(* Logix 5000 project; controller Almacen_1 vendor 1 type 14 code 235 rev 36.11; software revision 36.00 *)

TASK MainTask (continuous, watchdog 500 ms) : MainProgram, _02_Conveyor_1
TASK SafetyTask (periodic, rate 20 ms, priority 10, watchdog 20 ms, safety) : SafetyProgram

MODULES
   Local : vendor 1 type 14 code 235 (5069 0, rev 36.11)
      Logix_Principal : vendor 1 type 12 code 200 (Ethernet 10.12.143.10, rev 10.7, Output RPI 10 ms)
           Point_IO_Conveyor_1:2:I.4   // Sensor Piston Horizontal Extendido
           Point_IO_Conveyor_1:2:I.5   // Sensor Piston Horizontal Retraido
           Point_IO_Conveyor_1:2:I.6   // Sensor Inductivo Presencia en Zona de Vision (Actual Marcadora Laser)
           Point_IO_Conveyor_1:2:I.0   // Sensor difuso presencia lado B Almacen 2-1 (Robot)
           Point_IO_Conveyor_1:2:I.1   // Sensor difuso presencia lado B Almacen 2-2 (Robot)
           Point_IO_Conveyor_1:2:I.2   // Sensor Difuso Lado A CNC 3-1 (Centro-Marcadora Laser)
           Point_IO_Conveyor_1:2:I.3   // Sensor Difuso Lado A CNC 3-2 (Centro-Marcadora Laser)
           Point_IO_Conveyor_1:2:I.7   // Spare
           Point_IO_Conveyor_1:4:I.0   // Cambio de Dirección Extendido Lado A
           Point_IO_Conveyor_1:4:I.1   // Cambio de Dirección Retraido Lado A
           Point_IO_Conveyor_1:4:I.2   // Sensor 2 Posición Tope Corredizo Lado Almacen Izq
           Point_IO_Conveyor_1:4:I.3   // Sensor Inductivo Posición Lado B CNC
           Point_IO_Conveyor_1:4:I.6   // Sensor Límite Lado CNC Der
           Point_IO_Conveyor_1:4:I.7   // Sensor Posición Tope Corredizo Lado Almacen Der
           Point_IO_Conveyor_1:4:I.4   // Spare
           Point_IO_Conveyor_1:4:I.5   // Spare
           Point_IO_Conveyor_1:7:O.2   // Tope Piston CNC (Freno 5)
           Point_IO_Conveyor_1:7:O.3   // Tope Pison Marcadora Laser (Freno 06)
           Point_IO_Conveyor_1:7:O.4   // Subir Limit Switch
           Point_IO_Conveyor_1:7:O.5   // Tope Piston Cámara Visión
           Point_IO_Conveyor_1:7:O.6   // Sensor Límite Lado CNC Izq
           Point_IO_Conveyor_1:7:O.7   // Piston Cambio de Dirección Almacén
           Point_IO_Conveyor_1:7:O.0   // Piston Horizontal Para Salida de Pieza
           Point_IO_Conveyor_1:7:O.1   // Tope Piston Salida de Producto (Freno 8)
           Point_IO_Almacen1:2:I.5   // Boton Azul
           Point_IO_Almacen1:2:I.7   // Botón verde
           Point_IO_Almacen1:2:I.0   // Botón Verde Reset Vvula General Almacén 1
           Point_IO_Almacen1:3:O.0   // actuador posicionador horizontal lado derecho
           Point_IO_Almacen1:3:O.1   // actuador posicionador horizontal lado izquierdo
           Point_IO_Almacen1:3:O.2   // Actuador sencillo clamp abajo
           Point_IO_Almacen1:3:O.3   // Actuador Clamp arriba
           Point_IO_Almacen1:3:O.4   // actuador de giro direccion conveyor
           Point_IO_Almacen1:3:O.5   // actuador de giro direccion almacen
           Point_IO_Almacen1:3:O.6   // Posicion dejar pieza
           Point_IO_Almacen1:3:O.7   // Posicion tomar pieza
           Point_IO_Almacen1:4:O.0   // lampara LED verde botonera 1
           Point_IO_Almacen1:4:O.1   // RELEVADOR 1
           Point_IO_Almacen1:4:O.2   // RELEVADOR 2
           Point_IO_Almacen1:4:O.3   // RELEVADOR 3
           Point_IO_Almacen1:4:O.4   // RELEVADOR 4
           Point_IO_Almacen1:4:O.5   // RELEVADOR 5
           Point_IO_Almacen1:4:O.6   // RELEVADOR 6
           Point_IO_Almacen1:4:O.7   // SPARE
           Point_IO_Almacen1:5:O.0   // Luz Verde Almacen 1
           Point_IO_Almacen1:5:O.1   // Luz Ambar Almacen 1
           Point_IO_Almacen1:5:O.2   // Luz Roja Almacén 1
           Point_IO_Conveyor_1:1:I.2   // Boton negro Puerta
           Point_IO_Conveyor_1:1:I.3   // Boton Rojo Puerta
           Point_IO_Conveyor_1:1:I.4   // Auxiliar Scanner de Seguridad (Sin Conexión)
           Point_IO_Conveyor_1:1:I.6   // Sensor difuso presencia lado A Almacen 1-1
           Point_IO_Conveyor_1:1:I.7   // Sensor difuso presencia lado A Almacen 1-2
           Point_IO_Conveyor_1:1:I.0   // Spare
           Point_IO_Conveyor_1:1:I.1   // Spare
           Point_IO_Conveyor_1:1:I.5   // Spare
           Point_IO_Conveyor_1:3:I.2   // Sensor Piston Tope CNC
           Point_IO_Conveyor_1:3:I.3   // Sensor Piston Tope Marcadora Laser
           Point_IO_Conveyor_1:3:I.4   // Límit Switch Arriba
           Point_IO_Conveyor_1:3:I.5   // Sensor Piston Tope Camara Vision
           Point_IO_Conveyor_1:3:I.6   // Cambio de Dirección Extendido Lado B
           Point_IO_Conveyor_1:3:I.7   // Cambio de Dirección Retraido Lado B
           Point_IO_Conveyor_1:3:I.1   // Sensor Tope Piston Horizontal (Salida de conveyor)
           Point_IO_Conveyor_1:3:I.0   // Spare
           Point_IO_Conveyor_1:5:I.0   // Sensor Limit Switch Tope
           Point_IO_Conveyor_1:5:I.1   // Sensor Posición Tope Corredizo Lado Almacen Izq
           Point_IO_Conveyor_1:5:I.2   // Spare
           Point_IO_Conveyor_1:5:I.3   // Spare
           Point_IO_Conveyor_1:5:I.4   // Spare
           Point_IO_Conveyor_1:5:I.5   // Spare
           Point_IO_Conveyor_1:5:I.6   // Spare
           Point_IO_Conveyor_1:5:I.7   // Spare
           Point_IO_Conveyor_1:6:I.0   // Spare
           Point_IO_Conveyor_1:6:I.1   // Spare
           Point_IO_Conveyor_1:6:I.2   // Spare
           Point_IO_Conveyor_1:6:I.3   // Spare
           Point_IO_Conveyor_1:6:I.4   // Spare
           Point_IO_Conveyor_1:6:I.5   // Spare
           Point_IO_Conveyor_1:6:I.6   // Spare
           Point_IO_Conveyor_1:6:I.7   // Spare
           Point_IO_Conveyor_1:9:O.0   // Spare
           Point_IO_Conveyor_1:9:O.1   // Spare
           Point_IO_Conveyor_1:9:O.2   // Spare
           Point_IO_Conveyor_1:9:O.3   // Spare
           Point_IO_Conveyor_1:9:O.4   // Spare
           Point_IO_Conveyor_1:9:O.5   // Spare
           Point_IO_Conveyor_1:9:O.6   // Spare
           Point_IO_Conveyor_1:9:O.7   // Spare
           Point_IO_Conveyor_1:10:O.0   // Spare
           Point_IO_Conveyor_1:10:O.1   // Spare
           Point_IO_Conveyor_1:10:O.2   // Spare
           Point_IO_Conveyor_1:10:O.3   // Spare
           Point_IO_Conveyor_1:10:O.4   // Spare
           Point_IO_Conveyor_1:10:O.5   // Spare
           Point_IO_Conveyor_1:10:O.6   // Spare
           Point_IO_Conveyor_1:10:O.7   // Spare
           Point_IO_Conveyor_1:8:O.0   // Valvula Alimentacion de Aire Principal
           Point_IO_Conveyor_1:8:O.3   // Lampara Cognex 2
           Point_IO_Conveyor_1:8:O.4   // Lampara Cognex 1
           Point_IO_Conveyor_1:8:O.1   // Spare
           Point_IO_Conveyor_1:8:O.2   // Spare
           Point_IO_Conveyor_1:8:O.5   // Spare
           Point_IO_Conveyor_1:8:O.6   // Spare
           Point_IO_Conveyor_1:8:O.7   // Spare
         @c713d742@:Partner : vendor 1 type 14 code 146 (ICP 2, rev 31.11)
         PLC_Principal : vendor 1 type 14 code 148 (ICP 1, rev 31.11, $6ca47925$ RPI 15 ms, $8eacc5f3$ RPI 20 ms, $5ee93f34$ RPI 20 ms, $1738718a$ RPI 20 ms, $241c25b3$ RPI 20 ms)
      Conveyor_1 : PowerFlex 525-EENET (Ethernet 10.12.143.6, rev 5.1, Output RPI 20 ms)
      CognexGus : vendor 678 type 100 code 260 (Ethernet 10.12.143.155, rev 12.1, Output RPI 60 ms)
      Point_IO_Almacen1 : 1734-AENTR (Ethernet 10.12.143.40, rev 5.12, Output RPI 20 ms)
         E01N020S02 : 1734-IB8 (PointIO 2, rev 3.22)
         E01N020S01 : 1734-IB8 (PointIO 1, rev 3.22)
         E01NO20S03 : 1734-OB8 (PointIO 3, rev 3.22)
         E01N020S04 : 1734-OB8 (PointIO 4, rev 3.22)
         E01020S05 : 1734-OW4 (PointIO 5, rev 3.22)
         E01020S06 : vendor 1 type 35 code 15 (PointIO 6, rev 2.2, Input RPI 10 ms, Output RPI 20 ms)
         E01020S07 : vendor 1 type 35 code 16 (PointIO 7, rev 2.2, Input RPI 10 ms, Output RPI 20 ms)
      Point_IO_Conveyor_1 : 1734-AENTR (Ethernet 10.12.143.42, rev 5.12, Output RPI 20 ms)
         E01N022S01 : 1734-IB8 (PointIO 1, rev 3.22)
         E01N022S03 : 1734-IB8 (PointIO 3, rev 3.22)
         E01N022S05 : 1734-IB8 (PointIO 5, rev 3.22)
         E01N022S02 : 1734-IB8 (PointIO 2, rev 3.22)
         E01N022S04 : 1734-IB8 (PointIO 4, rev 3.22)
         E01N022S06 : 1734-IB8 (PointIO 6, rev 3.22)
         E01N022S08 : 1734-OB8 (PointIO 8, rev 3.22)
         E01N022S07 : 1734-OB8 (PointIO 7, rev 3.22)
         E01N022S10 : 1734-OW4 (PointIO 10, rev 3.22)
         E01N022S09 : 1734-OW4 (PointIO 9, rev 3.22)
         E01N022S011 : vendor 1 type 35 code 15 (PointIO 11, rev 2.2, Input RPI 10 ms, Output RPI 20 ms)
              Point_IO_Conveyor_1:11:I.Pt03Data   // Spare
              Point_IO_Conveyor_1:11:I.Pt01Data   // E_Stop Conveyor 1 Presionado
              Point_IO_Conveyor_1:11:I.Pt04Data   // Spare
              Point_IO_Conveyor_1:11:I.Pt02Data   // Spare
              Point_IO_Conveyor_1:11:I.Pt06Data   // Spare
              Point_IO_Conveyor_1:11:I.Pt00Data   // E_Stop Conveyor 1 Liberado
              Point_IO_Conveyor_1:11:I.Pt07Data   // Spare
              Point_IO_Conveyor_1:11:I.Pt05Data   // Spare
         E01N022S12 : vendor 1 type 35 code 16 (PointIO 12, rev 2.2, Input RPI 10 ms, Output RPI 20 ms)
              Point_IO_Conveyor_1:12:O.Pt01Data   // S2 PowerFlex Transportador 1
              Point_IO_Conveyor_1:12:O.Pt04Data   // Spare
              Point_IO_Conveyor_1:12:O.Pt03Data   // Spare
              Point_IO_Conveyor_1:12:O.Pt07Data   // Spare
              Point_IO_Conveyor_1:12:O.Pt05Data   // Spare
              Point_IO_Conveyor_1:12:O.Pt02Data   // Spare
              Point_IO_Conveyor_1:12:O.Pt06Data   // Spare
              Point_IO_Conveyor_1:12:O.Pt00Data   // S1 PowerFlex Transportador 1
END_MODULES

ADD_ON_INSTRUCTION Debounce   (* revision 1.0, vendor Premier Tech Ltd, ExecuteEnableInFalse *)
// Revision note:
// 1.0 Master 1st release
VAR_INPUT
   FilterOnTimerPreset : ALIAS FOR FilterOnTimer.PRE; {required}   // Digital input filter time preset (ON)
   FilterOffTimerPreset : ALIAS FOR FilterOffTimer.PRE; {required}   // Digital input filter time preset (OFF)
END_VAR
VAR_OUTPUT
   B : BOOL; {access Read Only, visible}   // Digital input filtered signal
   BFT : BOOL; {access Read Only}   // Falling transient: digital input filtered signal
   BRT : BOOL; {access Read Only}   // Rising transient: digital input filtered signal
   I : BOOL; {access Read Only}   // Digital input raw signal
   IFT : BOOL; {access Read Only}   // Falling transient: digital input raw signal
   IRT : BOOL; {access Read Only}   // Rising transient: digital input raw signal
END_VAR
VAR
   FilterOffTimer : TIMER;   // Digital input filter time (OFF)
   FilterOnTimer : TIMER;   // Digital input filter time (ON)
   B_Osr : BOOL; {access None}
   B_Osf : BOOL; {access None}
   I_Osr : BOOL; {access None}
   I_Osf : BOOL; {access None}
END_VAR

ROUTINE EnableInFalse   (* ladder *)
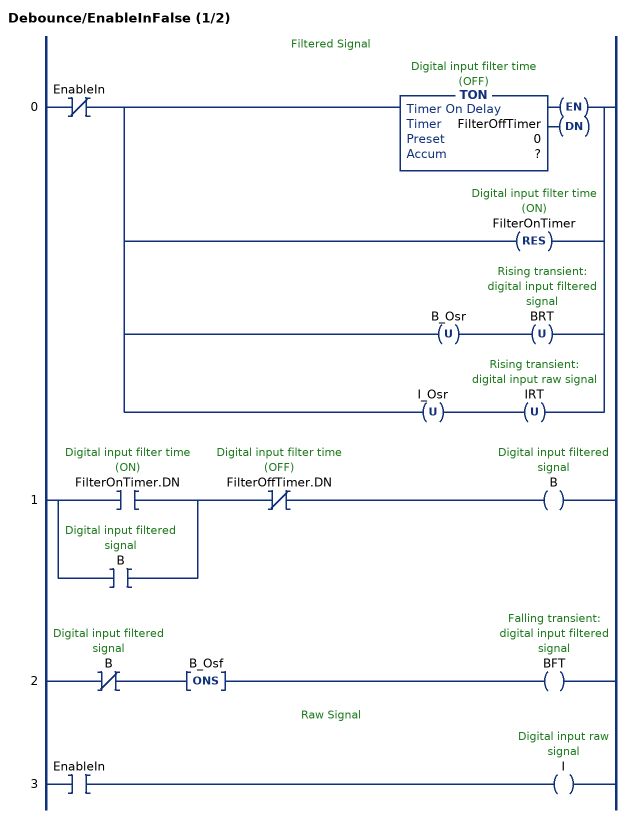
   // Filtered Signal
   0: XIO(EnableIn)[TON(FilterOffTimer,?,?) ,RES(FilterOnTimer) ,OTU(B_Osr) OTU(BRT) ,OTU(I_Osr) OTU(IRT) ];
   1: [XIC(FilterOnTimer.DN) ,XIC(B) ]XIO(FilterOffTimer.DN)OTE(B);
   2: XIO(B)ONS(B_Osf)OTE(BFT);
   // Raw Signal
   3: XIC(EnableIn)OTE(I);
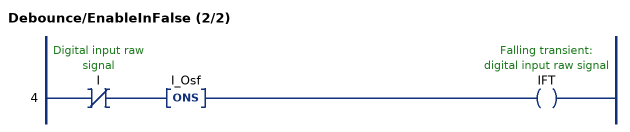
   4: XIO(I)ONS(I_Osf)OTE(IFT);
END_ROUTINE

ROUTINE Logic   (* ladder *)
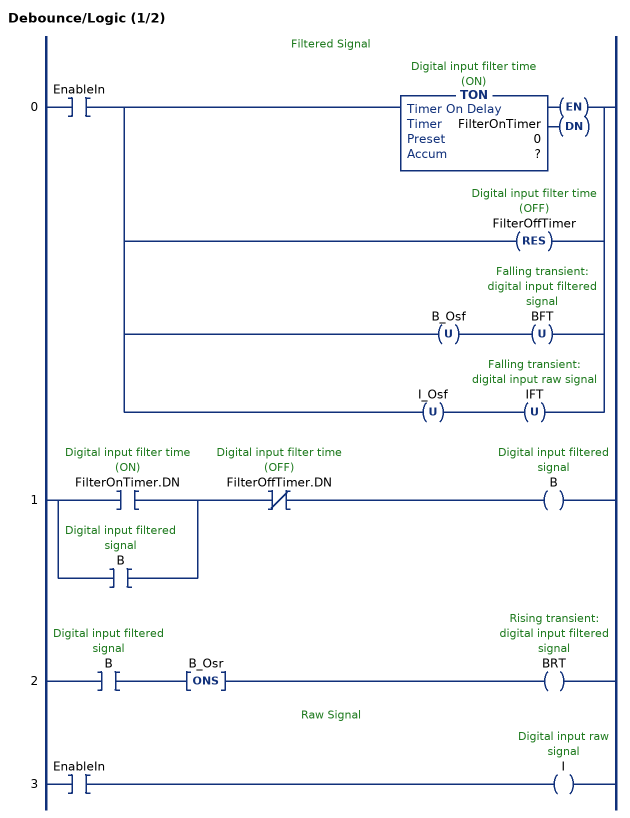
   // Filtered Signal
   0: XIC(EnableIn)[TON(FilterOnTimer,?,?) ,RES(FilterOffTimer) ,OTU(B_Osf) OTU(BFT) ,OTU(I_Osf) OTU(IFT) ];
   1: [XIC(FilterOnTimer.DN) ,XIC(B) ]XIO(FilterOffTimer.DN)OTE(B);
   2: XIC(B)ONS(B_Osr)OTE(BRT);
   // Raw Signal
   3: XIC(EnableIn)OTE(I);
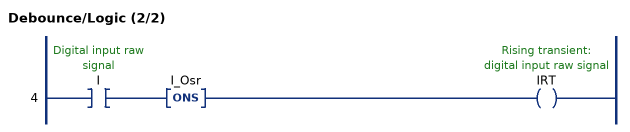
   4: XIC(I)ONS(I_Osr)OTE(IRT);
END_ROUTINE
END_ADD_ON_INSTRUCTION

VAR_GLOBAL   (* controller tags *)
   Alarms_OK : BOOL := 1;
   Alm1_GripperClosed : BOOL;
   Alm1_GripperOpen : BOOL := 1;
   Alm1_S1 : BOOL;
   Alm1_S2 : BOOL;
   Alm1_X1 : BOOL;
   Alm1_X2 : BOOL := 1;
   Alm1_Z1 : BOOL;
   Alm1_Z2 : BOOL;
   Alm2_Home : BOOL;
   AlmPosReq : DINT;
   Altura_Servo : DINT;
   At_Pos_Alm_1 : DINT := 8;
   Auto_Conv_1 : BOOL := 1;   // Secuencia Activada Automática Conveyor 1
   Auto_Enabled : BOOL;
   Bit_CambioDir_Conv_1 : BOOL;
   Bit_CambioDirAlm_Conv_1 : BOOL;
   Bit_FinDeCarreraConv_1 : BOOL;
   Bit_Reset_ValvulaGeneral_Conv_1 : BOOL;
   Bit_Reset_ValvulaGeneral_Conv_2 : BOOL := 1;
   Bit_Salida_Mat_Conv_1 : BOOL;   // Bit de Retorno de pieza a Almacen Conveyor 1
   Btn_Negro_Conv_1 : BOOL;   // Botón Negro Puerta de Conveyor 1
   Btn_Negro_Conv_2 : BOOL;   // Botón Negro Puerta de Conveyor 2
   Btn_Rojo_Conv_1 : BOOL;   // Botón Rojo Puerta de Conveyor 1
   Btn_Rojo_Conv_2 : BOOL;   // Botón Rojo Puerta de Conveyor 2
   CambioDir_Ext_Almacen_Conv_1 : BOOL;   // Sensor Cambio de Dirección Extendido Lado A (Almacén)
   CambioDir_Ext_Almacen_Conv_2 : BOOL;   // Sensor Cambio de Dirección Extendido Lado A Almacén
   CambioDir_Ext_CNC_Conv_1 : BOOL;   // Sensor Cambio de Dirección Extendido Lado B (CNC)
   CambioDir_Ext_CNC_Conv_2 : BOOL;   // Cambio de Dirección Extendido Lado B CNC
   CambioDir_Ret_Almacen_Conv_1 : BOOL := 1;   // Sensor Cambio de Dirección Retraido Lado A (Almacén)
   CambioDir_Ret_Almacen_Conv_2 : BOOL;   // Sensor Cambio de Dirección Retraido Lado A Almacén
   CambioDir_Ret_CNC_Conv_1 : BOOL;   // Sensor Cambio de Dirección Retraido Lado B (CNC)
   CambioDir_Ret_CNC_Conv_2 : BOOL;   // Cambio de Dirección Retraido Lado B CNC
   Carro_A : BOOL := 1;
   Carro_B : BOOL;
   Carro_C : BOOL;
   Carro_D : BOOL;
   Carro_E : BOOL;
   Carro_F : BOOL;
   Carro_G : BOOL;
   Carro_H : BOOL;
   Carro_I : BOOL;
   Carro_J : BOOL;
   Carro_Posicion_X_Negativo : BOOL;   // Posición del Carro Cercano al Almacén1 Almacén 1
   Carro_Posicion_X_Positivo : BOOL := 1;   // Posición del Carro Cercano al Conveyor 1 Almacén 1
   Carro_Posicion_Y_Negativo : BOOL;   // Posición Carro a la Derecha Área de Salidas Almacén 1
   Carro_Posicion_Y_Positivo : BOOL;   // Posición Carro a la Izquierda Área de Entradas Almacén 1
   Carro_Posicion_Yaw_Negativo : BOOL;   // Giro Dirección Almacén Almacén 1
   Carro_Posicion_Yaw_Positivo : BOOL;   // Giro Dirección Conveyor Almacén 1
   Carro_Posicion_Z_Negativo : BOOL;   // Presionar Pieza Almacén 1
   Carro_Posicion_Z_Positivo : BOOL := 1;   // Soltar Pieza Almacén 1
   CellAuto : BOOL;
   Cmd_CloseGripper_Alm1 : BOOL;
   Cmd_OpenGripper_Alm1 : BOOL;
   Cmd_StorageHome_Alm1 : BOOL;
   Cmd_StoS1Pos_Alm1 : BOOL;   // Giro Lado de Almacén 2
   Cmd_StoS2Pos_Alm1 : BOOL;   // Giro Lado de Conveyor 2
   Cmd_XtoX1Pos_Alm1 : BOOL;   // Lado Entrada almacén 2
   Cmd_XtoX2Pos_Alm1 : BOOL;   // Lado Salida Almacén 2
   Cmd_YPickSafe_Alm1 : BOOL;
   Cmd_YPlaceSAfe_Alm1 : BOOL;
   Cmd_YtoYOff_Alm1 : BOOL;
   Cmd_YtoYPick_Alm1 : BOOL;
   Cmd_YtoYPlace_Alm1 : BOOL;
   Cmd_YtoYPlaceOffset_Alm1 : BOOL;
   Cmd_ZtoZ1Pos_Alm1 : BOOL;   // Lado del Conveyor 2
   Cmd_ZtoZ2Pos_Alm1 : BOOL;   // Lado del Almacén 2
   Consumed_Signals_TEC_81_Conveyor_1 : DINT;
   Continuar_Secuencia_en_Conveyor_1 : BOOL;   // Bit de Terminación de Procesos de CNC 1 y Mesa KUKA
   Conv_1_ON : BOOL;
   Conv_1_Vacio_Inicial : BOOL := 1;   // Bit de Verificación Conveyor 1 Vacio
   Debounce_Alimentacion_Conv_1 : Debounce;
   Debounce_Almacen_Conv_1 : Debounce;
   Debounce_CNC_2_Conv_1 : Debounce;
   Debounce_CNC_Conv_1 : Debounce;
   Debounce_Entrada_Conv_1 : Debounce;
   Debounce_Marcadora_Conv_1 : Debounce;
   Done_Step_00_Alm_1 : BOOL;
   Done_Step_00_Conv_1 : BOOL;
   Done_Step_01_Alm_1 : BOOL;
   Done_Step_01_Conv_1 : BOOL;
   Done_Step_02_Alm_1 : BOOL;
   Done_Step_02_Conv_1 : BOOL;
   Done_Step_03_Alm_1 : BOOL;
   Done_Step_03_Conv_1 : BOOL;
   Done_Step_04_A_Conv_1 : BOOL;
   Done_Step_04_Alm_1 : BOOL;
   Done_Step_04_Conv_1 : BOOL;
   Done_Step_05_Alm_1 : BOOL;
   Done_Step_05_Conv_1 : BOOL;
   Done_Step_06_Alm_1 : BOOL;
   Done_Step_06_Conv_1 : BOOL;
   Done_Step_07_Alm_1 : BOOL;
   Done_Step_07_Conv_1 : BOOL;
   Done_Step_08_Alm_1 : BOOL;
   Done_Step_08_Conv_1 : BOOL;
   Done_Step_09_Alm_1 : BOOL;
   Done_Step_09_Conv_1 : BOOL;
   Done_Step_10_Alm_1 : BOOL;
   Done_Step_10_Conv_1 : BOOL;
   Done_Step_11_Alm_1 : BOOL;
   Done_Step_11_Conv_1 : BOOL;
   Done_Step_12_Alm_1 : BOOL;
   Done_Step_12_Conv_1 : BOOL;
   Done_Step_13_Alm_1 : BOOL;
   Done_Step_13_Conv_1 : BOOL;
   Done_Step_14_Alm_1 : BOOL;
   Done_Step_14_Conv_1 : BOOL;
   Done_Step_15_Alm_1 : BOOL;
   Done_Step_15_Conv_1 : BOOL;
   Done_Step_16_Alm_1 : BOOL;
   Done_Step_16_Conv_1 : BOOL;
   Done_Step_17_Alm_1 : BOOL;
   Done_Step_17_Conv_1 : BOOL;
   Done_Step_18_Alm_1 : BOOL;
   Done_Step_18_Conv_1 : BOOL;
   Done_Step_19_Alm_1 : BOOL;
   Done_Step_19_Conv_1 : BOOL;
   Done_Step_20_Alm_1 : BOOL;
   Done_Step_20_Conv_1 : BOOL;
   Done_Step_21_Alm_1 : BOOL;
   Done_Step_21_Conv_1 : BOOL;
   Done_Step_22_Alm_1 : BOOL;
   Done_Step_22_Conv_1 : BOOL;
   Done_Step_23_Conv_1 : BOOL;
   Done_Step_24_Conv_1 : BOOL;
   Done_Step_25_Conv_1 : BOOL;
   Done_Step_26_Conv_1 : BOOL;
   Done_Step_27_Conv_1 : BOOL;
   Done_Step_28_Conv_1 : BOOL;
   Done_Step_29_Conv_1 : BOOL;
   Done_Step_30_Conv_1 : BOOL;
   Done_Step_31_Conv_1 : BOOL;
   Done_Step_32_Conv_1 : BOOL;
   Done_Step_33_Conv_1 : BOOL;
   Done_Step_34_Conv_1 : BOOL;
   Done_Step_35_Conv_1 : BOOL;
   Done_Step_36_Conv_1 : BOOL;
   Done_Step_37_Conv_1 : BOOL;
   Done_Step_38_Conv_1 : BOOL;
   Done_Step_39_Conv_1 : BOOL;
   Done_Step_40_Conv_1 : BOOL;
   End_Alm_Start_Conv : BOOL;   // Almacén Entrega Pieza a Conveyor
   End_Conv_Start_Alm : BOOL;   // Termina Conveyor Empieza Almacén Con Pieza Terminada
   EStops_OK : BOOL;
   EStops_OK_External_A1 : DINT := 3;
   Fanuc_Griper_Cerrado_Conv_1 : BOOL := 1;   // Señal desde Robot Fanuc Para indicar el Cerrado de Griper Exclusivo Conveyor 1
   Fanuc_Posicion_Dejar_Pieza_Conv_1 : BOOL;   // Señal del Robot Fanuc de confirmación de Dejar Pieza en Conveyor 1
   Fanuc_Posicion_Dejar_Pieza_Mesa_1 : BOOL := 1;   // Señal de Posición del Robot Fanuc para dejar Pieza en Pistón 1 de la Mesa Kuka Conveyor 1
   Fanuc_Posicion_Segura_CNC_1 : BOOL := 1;   // Posición Segura de Robot Fanuc Después de Dejar Pieza en CNC 1 Conveyor 1
   Fanuc_Posicion_Segura_Mesa_1 : BOOL := 1;   // Posición Segura Frente a Mesa Kuka Conveyor 1
   Fanuc_RetornoPieza_Conv_1 : BOOL;   // Señal de Robot Fanuc Retorno de Pieza después de CNC
   Fixture_Sensor_Direccion_Conveyor : BOOL;   // Señal del Almacén de que el Fisture está listo para Tomar Pieza a la salida
   Green_Light_Alm_1 : BOOL;
   Green_Light_Alm_2 : BOOL := 1;
   Griper_Down : BOOL;
   Griper_Up : BOOL := 1;
   HMI_Almacen_In : DINT;
   HMI_Almacen_Reset_Sequence : BOOL;   // Restablece Secuencia de Almacén al Paso Inicial
   HMI_Conveyor_Reset_Sequence : BOOL;   // Restablece Secuencia de Conveyor al Paso Inicial
   HMI_Conveyor_Select_Sequence : BOOL;   // Prueba Para seleccionar Paso
   HMI_Conveyor_Start : BOOL;   // Botón HMI para Empezar Secuencia
   HMI_Reset_PowerFlex525 : BOOL;
   HMI_Start : BOOL;
   HomeSeq : DINT;
   HomeStep0 : BOOL := 1;   // Request for Home
   HomeStep1 : BOOL;   // Evaluar Condiones a seguir
   HomeStep2 : BOOL;   // S to S1
   HomeStep3 : BOOL;   // S to S2
   HomeStep4 : BOOL;   // Y to Y Home
   HomeStep5 : BOOL;   // Z to Z1
   HomeStep6 : BOOL;   // S to S1
   HomeStep7 : BOOL;   // X to X1
   HomeStep8 : BOOL;   // Open Gripper
   Homestep9 : BOOL;   // Homed
   HomeStorageDone : BOOL;
   HomeStorageRequired : BOOL := 1;
   HomeStoSeqToTec81_Alm1 : DINT; {produced}
   HommingCycle : BOOL;
   HommingStorage : BOOL;
   In_Pos_Alm_1 : DINT;
   IndexPickStorage2 : DINT := 1;
   Inicializacion_FirstShot : BOOL := 1;   // Bit Para Limpiar Datos al Inicio de Programa
   InicioCiclo : BOOL;
   KUKA_Posicion_Segura : BOOL := 1;   // Posición Segura del Robot KUKA Sin Movimiento, en Espera de Recibir Pieza
   KUKA_Proceso_Terminado_Conv_1 : BOOL;   // Proceso Terminado para Pieza de Conveyor 1
   Limit_UP_Conv_1 : BOOL;   // Subir Limit Switch Conveyor 1
   Limit_UP_Conv_2 : BOOL;   // Subir Limit Switch Conveyor 2
   M1 : BOOL;
   M10 : BOOL;
   M11 : BOOL;
   M12 : BOOL;
   M13 : BOOL;
   M14 : BOOL := 1;
   M15 : BOOL;
   M16 : BOOL := 1;
   M2 : BOOL;
   M3 : BOOL;
   M4 : BOOL;
   M5 : BOOL;
   M6 : BOOL;
   M7 : BOOL;
   M8 : BOOL := 1;
   M9 : BOOL;
   MainSeq : DINT;
   Manual_Conv_1 : BOOL;   // Secuencia Activada Manual Conveyor 1
   Memory : BOOL;
   Mesa_Kuka_Piston_1_Abierto : BOOL := 1;   // Pistón Para Sujetar Pieza de conveyor 1 Abierta Conveyor 1
   ONS_Marcadora : BOOL;
   Permissive_HomeStep0 : BOOL;
   Permissive_homeStep1 : BOOL;
   Permissive_HomeStep2 : BOOL;
   Permissive_HomeStep3 : BOOL;
   Permissive_HomeStep4 : BOOL;
   Permissive_HomeStep5 : BOOL;
   Permissive_HomeStep6 : BOOL;
   Permissive_HomeStep7 : BOOL;
   Permissive_HomeStep8 : BOOL;
   Permissive_HomeStep9 : BOOL;
   Permissive_Step0 : BOOL;
   Permissive_Step1 : BOOL;
   Permissive_Step10 : BOOL;
   Permissive_Step11 : BOOL;
   Permissive_Step12 : BOOL;
   Permissive_Step13 : BOOL;
   Permissive_Step14 : BOOL;
   Permissive_Step15 : BOOL;
   Permissive_Step16 : BOOL;
   Permissive_Step17 : BOOL;
   Permissive_Step18 : BOOL;
   Permissive_Step19 : BOOL;
   Permissive_Step2 : BOOL;
   Permissive_Step20 : BOOL;
   Permissive_Step21 : BOOL;
   Permissive_Step22 : BOOL;
   Permissive_Step23 : BOOL;
   Permissive_Step24 : BOOL;
   Permissive_Step25 : BOOL;
   Permissive_Step26 : BOOL;
   Permissive_Step3 : BOOL;
   Permissive_Step4 : BOOL;
   Permissive_Step5 : BOOL;
   Permissive_Step6 : BOOL;
   Permissive_Step7 : BOOL;
   Permissive_Step8 : BOOL;
   Permissive_Step9 : BOOL;
   PF_ClearFault_525_Conv_1 : BOOL;   // Clear Fault PowerFlex Conveyor 1
   PF_On_525_Conv_1 : BOOL;   // Encender/Apagar PowerFlex Conveyor 1
   PickPosition_Alm_1 : Position_Storage;
   PickPositionProd_Alm1 : Position_Storage; {produced}
   Piston_CambioDir_Almacen_Conv_1 : BOOL;   // Cambiar Direccion de Pieza Lado Almacen Conveyor 1
   Piston_CambioDir_Almacen_Conv_2 : BOOL;   // Cambiar Direccion de Pieza Lado Almacen Conveyor 2
   Piston_CambioDir_CNC_Conv_1 : BOOL;   // Cambiar Dirección de Pieza Lado CNC Conveyor 1
   Piston_CambioDir_CNC_Conv_2 : BOOL;   // Cambiar Dirección de Pieza Lado CNC Conveyor 2
   Piston_Horizontal_Conv_1 : BOOL;   // Extender Pistón Horizontal del Conveyor 1
   Piston_Horizontal_Conv_2 : BOOL;   // Extender Pistón Horizontal del Conveyor 2
   PlacePosition : Position_Storage;
   PlacesStorage2 : Position_Storage[20];
   PosicionAlmacen : DINT := 1;
   Prensa_Abierta_CNC_1 : BOOL := 1;   // Sensor para Detectar Prensa Abierta CNC 1 Conveyor 1
   Prensa_Presencia_Pieza_CNC_1 : BOOL := 1;   // Sensor para detectar Pieza dentro de la Prensa del CNC 1 Conveyor 1
   Presencia_TomaFanuc_Conv_1 : BOOL;   // Presencia de Pieza Ubicada en Área para Tomar del Robot Fanuc (CNC)
   Produced_Signals_Conveyor_1_TEC_81 : DINT := 256; {produced}   // Arreglo de Tags Enviadas del Conveyor 1 al Robot Fanuc
   Puerta_Abierta_CNC_1 : BOOL := 1;   // Sensor de Puerta Abierta en CNC 1 Conveyor 1
   PV_Auto : BOOL := 1;
   PV_Hold : BOOL;
   PV_HomeStorage : BOOL;
   PV_SelectedPlace : BOOL;
   PV_Start : BOOL;
   PV_UndoSelect : BOOL;
   Red_Light_Alm_1 : BOOL := 1;
   Red_Light_Alm_2 : BOOL;
   Resert_PF525_From_SFTY : DINT;
   Reset_Almacen_1_PF525_Conv_1 : BOOL;
   Reset_Almacen_2_PF525_Conv_2 : BOOL;
   Reset_PF_Conv_1 : BOOL;
   Reset_ValvulaGeneral_Conv_1 : BOOL;
   Reset_ValvulaGeneral_Conv_2 : BOOL;
   RunningCycle : BOOL;
   Safety_OK : BOOL;
   Secuencia_Finalizada_Conv_1 : BOOL;
   Secuencia_Iniciada_Conv_1 : BOOL;
   Sensor_Difuso_1_1_Conv_1 : BOOL;   // Sensor Lado A Almacen 1-1
   Sensor_Difuso_1_1_Conv_2 : BOOL;   // Sensor Difuso Presencia Lado A Almacen 1-1
   Sensor_Difuso_1_2_Conv_1 : BOOL;   // Sensor Lado A Almacen 1-2
   Sensor_Difuso_1_2_Conv_2 : BOOL;   // Sensor Difuso Presencia Lado A Almacén 1-2
   Sensor_Difuso_2_1_Conv_1 : BOOL;   // Sensor Lado B Almacen 2-1
   Sensor_Difuso_2_1_Conv_2 : BOOL;   // Sensor Difuso Presencia Lado B CNC 2-1
   Sensor_Difuso_2_2_Conv_1 : BOOL;   // Sensor Lado B Almacen 2-2
   Sensor_Difuso_2_2_Conv_2 : BOOL;   // Sensor Difuso Presencia Lado B CNC 2-2
   Sensor_Difuso_3_1_Conv_1 : BOOL;   // Sensor Lado A CNC 3-1
   Sensor_Difuso_3_1_Conv_2 : BOOL;   // Sensor Difuso Presencia Lado A CNC 3-1
   Sensor_Difuso_3_2_Conv_1 : BOOL;   // Sensor Lado A CNC 3-2
   Sensor_Difuso_3_2_Conv_2 : BOOL;   // Sensor Difuso Presencia Lado A CNC 3-2
   Sensor_Inductivo_Alimentacion_Conv_1 : BOOL;   // Sensor Inductivo Alimentacion y Salida Almacen Conveyor 1
   Sensor_Inductivo_Almacen_Conv_1 : BOOL;   // Sensor Inductivo Lado A Final derecha Almacen
   Sensor_Inductivo_Almacen_Conv_2 : BOOL;   // Sensor Inductivo Lado A Almacén (Entrada)
   Sensor_Inductivo_CNC_2_Conv_1 : BOOL;   // Sensor Inductivo Lado B CNC
   Sensor_Inductivo_CNC_2_Conv_2 : BOOL;   // Sensor Inductivo Posición Lado A CNC
   Sensor_Inductivo_CNC_Conv_1 : BOOL;   // Sensor Inductivo Lado A CNC
   Sensor_Inductivo_CNC_Conv_2 : BOOL;   // Sensor Inductivo Posición Lado B CNC
   Sensor_Inductivo_Entrada_Conv_1 : BOOL;   // Sensor Inductivo Entrada Lado CNC (Adelante)
   Sensor_Inductivo_Entrada_Conv_2 : BOOL;   // Sensor Inductivo Lado B CNC (Entrada) Conveyor 2
   Sensor_Inductivo_Limit_Conv_2 : BOOL;   // Sensor Inductivo Limit Switch (Revisarl, Empate)
   Sensor_Inductivo_Marcadora_Conv_1 : BOOL;   // Sensor Inductivo Presencia Zona Marcadora Laser
   Sensor_Inductivo_Salida_Conv_2 : BOOL;   // Sensor Inductivo a Salida/entrada Almacen
   Sensor_Inductivo_Vision_Conv_2 : BOOL;   // Sensor Presencia Zona de Marcadora Láser
   Sensor_Limit_Up_Conv_1 : BOOL;   // Limit Switch Arriba
   Sensor_Limit_Up_Conv_2 : BOOL;   // Limit Switch Arriba
   Sensor_PH_Ext_Conv_1 : BOOL;   // Sensor Pistón Horizontal Extendido
   Sensor_PH_Ret_Conv_1 : BOOL := 1;   // Sensor Pistón Horizontal Retraido
   Sensor_PistHor_Ext_Conv_2 : BOOL;   // Sensor Pistón Horizontal Extendido
   Sensor_PistHor_Ret_Conv_2 : BOOL;   // Sensor Pistón Horizontal Retraido
   Sensor_Tope_CNC_Conv_1 : BOOL;   // Sensor Pistón Tope CNC
   Sensor_Tope_CNC_Conv_2 : BOOL;   // Sensor Tope Pistón CNC
   Sensor_Tope_Marcadora_Conv_1 : BOOL;   // Sensor Pistón Tope Marcadora Láser
   Sensor_Tope_Marcadora_Conv_2 : BOOL;   // Sensor Pistón Tope Marcadora Láser
   Sensor_Tope_PH_Conv_1 : BOOL;   // Sensor Tope Pistón Horizontal
   Sensor_Tope_PH_Conv_2 : BOOL;   // Sensor Tope Pistón Horizontal (Salida de Conveyor 2)
   Sensor_Tope_Vision_Conv_1 : BOOL;   // Sensor Pistón Tope Cámara de Visión
   Sensor_Tope_Vision_Conv_2 : BOOL;   // Sensor Pistón Tope Cámara de Visión
   Sequence_Mover_A_Marcadora_Conv_1 : BOOL;   // Secuencia de Salida de Producto Maquinado Cambiar a Marcadora Laser
   Sequence_MoverACamara_Conv_1 : BOOL;   // Secuencia de Movimiento de PF525 Hasta posición de Cámara
   Sequence_Start_Conv_1 : BOOL;   // Inicia Secuenca Automática Lleva Pieza a Toma Fanuc Conveyor 1
   Signal_CNC_1_Abrir_Prensa_Conv_1 : BOOL;   // Señal para Abrir Prensa en CNC 1
   Signal_CNC_1_Cerrar_Prensa_Conv_1 : BOOL;   // Señal para cerrar Prensa en CNC 1
   Signal_CNC_1_Cerrar_Puerta_Conv_1 : BOOL;   // Señal para cerrar la puerta del CNC 1 Conveyor 1
   Signal_Fanuc_Acercar_MesaKuka_Conv_1 : BOOL;   // Señal para Acercar al Robot Fanuc a posición del Pistón de la Mesa Kuka Conveyor 1
   Signal_Fanuc_Acercar_Pieza_CNC_Conv_1 : BOOL;   // Robot Fanuc Acerca pieza a CNC y la posiciona en la prensa
   Signal_Fanuc_Dejar_MesaKuka_Conv_1 : BOOL;   // Señal para Robot Fanuc de Dejar pieza en Mesa Kuka y moverse a posición segura
   Signal_Fanuc_Dejar_Pieza_CNC_Conv_1 : BOOL;   // Robot Fanuc suelta la pieza dentro del CNC una vez que la prensa la está sujetando y se mueve a posición segura
   Signal_Fanuc_Dejar_Pieza_Conv_1 : BOOL := 1;   // Señal para Robot Fanuc de moverse y Dejar Pieza en Conveyor 1
   Signal_Fanuc_Mover_MesaKuka_Conv_1 : BOOL;   // Señal para Mover el Robot Fanuc a posición segura frente a Mesa KUKA
   Signal_Fanuc_Sujetar_MesaKuka_Conv_1 : BOOL;   // Señal para Robot Fanuc para Sujetar Pieza en Mesa Kuka sin moverse Conveyor 1
   Signal_Fanuc_Sujetar_Pieza_CNC_Conv_1 : BOOL;   // Robot Fanuc se acerca a la Pieza dentro de CNC 1 y la sujeta Espera señal para moverse
   Signal_Fanuc_Tomar_Pieza_Conv_1 : BOOL;   // Señal para Tomar pieza desde el Conveyor 1 Hacia CNC
   Signal_Marcadora_Conv_1 : BOOL;   // Señal Para encender la Marcadora
   Signal_MesaKuka_Abrir_Piston_Conv_1 : BOOL;   // Señal para Abrir Pistón en Mesa Kuka Conveyor 1
   Signal_MesaKuka_Cerrar_Piston_Conv_1 : BOOL;   // Señal para Cerrar Pistón en la Mesa Kuka Conveyor 1
   Signal_MesaKuka_Iniciar_Proceso_Conv_1 : BOOL;   // Señal para Robot Kuka de iniciar proceso de Acabado
   Slector_Automatico_Conv_1 : BOOL := 1;   // Bit Selector Automático ON
   Start_Almacen_1_PF525_Conv_1 : BOOL;   // Inicializa o Arranca el Conveyor 1 PF525
   Start_Kinetix_Alm_1 : DINT; {produced}
   Start_Motor_Alm_1 : BOOL;
   Step0 : BOOL := 1;   // Condiciones iniciales
   Step1 : BOOL;   // Y to Y Pick
   Step10 : BOOL;   // Open Gripper
   Step11 : BOOL;   // Y to Y place safe
   step12 : BOOL;   // Z to Z2
   step13 : BOOL;   // Esperar Pieza Terminada
   Step14 : BOOL;   // Y to Y place
   Step15 : BOOL;   // Z to Z1
   Step16 : BOOL;   // Close Gripper
   Step17 : BOOL;   // Y to Y PlaceOffset
   Step18 : BOOL;   // S t o S1
   Step19 : BOOL;   // X to X2
   Step2 : BOOL;   // X to X1
   Step20 : BOOL;   // Y to Y PickOffset
   Step21 : BOOL;   // Z to Z2
   Step22 : BOOL;   // Y to Y Pick
   Step23 : BOOL;   // Open Gripper
   Step24 : BOOL;   // Y to Y Pcik Safe
   Step25 : BOOL;   // Z to Z1
   Step26 : BOOL;   // Homming
   Step3 : BOOL;   // Z to Z2
   Step4 : BOOL;   // Close Gripper
   Step5 : BOOL;   // Y to Y PickOffset
   Step6 : BOOL;   // Z to Z1
   Step7 : BOOL;   // Y to Y PlaceOffset
   Step8 : BOOL;   // S to S2
   step9 : BOOL;   // Y to Y Place
   Step_00_Alm_1 : BOOL := 1;
   Step_00_Conv_1 : BOOL;
   Step_01_Alm_1 : BOOL;
   Step_01_Conv_1 : BOOL;
   Step_02_Alm_1 : BOOL;
   Step_02_Conv_1 : BOOL;
   Step_03_Alm_1 : BOOL;
   Step_03_Conv_1 : BOOL;
   Step_04_Alm_1 : BOOL;
   Step_04_Conv_1 : BOOL;
   Step_05_Alm_1 : BOOL;
   Step_05_Conv_1 : BOOL;
   Step_06_Alm_1 : BOOL;
   Step_06_Conv_1 : BOOL;
   Step_07_Alm_1 : BOOL;
   Step_07_Conv_1 : BOOL;
   Step_08_Alm_1 : BOOL;
   Step_08_Conv_1 : BOOL;
   Step_09_Alm_1 : BOOL;
   Step_09_Conv_1 : BOOL;
   Step_10_Alm_1 : BOOL;
   Step_10_Conv_1 : BOOL;
   Step_11_Alm_1 : BOOL;
   Step_11_Conv_1 : BOOL;
   Step_12_Alm_1 : BOOL;
   Step_12_Conv_1 : BOOL;
   Step_13_Alm_1 : BOOL;
   Step_13_Conv_1 : BOOL;
   Step_14_Alm_1 : BOOL;
   Step_14_Conv_1 : BOOL;
   Step_15_Alm_1 : BOOL;
   Step_15_Conv_1 : BOOL;
   Step_16_Alm_1 : BOOL;
   Step_16_Conv_1 : BOOL;
   Step_17_Alm_1 : BOOL;
   Step_17_Conv_1 : BOOL;
   Step_18_Alm_1 : BOOL;
   Step_18_Conv_1 : BOOL;
   Step_19_Alm_1 : BOOL;
   Step_19_Conv_1 : BOOL;
   Step_20_Alm_1 : BOOL;
   Step_20_Conv_1 : BOOL;
   Step_21_Alm_1 : BOOL;
   Step_21_Conv_1 : BOOL;
   Step_22_Alm_1 : BOOL;
   Step_22_Conv_1 : BOOL;
   Step_23_Conv_1 : BOOL;
   Step_24_Conv_1 : BOOL := 1;
   Step_25_Conv_1 : BOOL;
   Step_26_Conv_1 : BOOL;
   Step_27_Conv_1 : BOOL;
   Step_28_Conv_1 : BOOL;
   Step_29_Conv_1 : BOOL;
   Step_30_Conv_1 : BOOL;
   Step_31_Conv_1 : BOOL;
   Step_32_Conv_1 : BOOL;
   Step_33_Conv_1 : BOOL;
   Step_34_Conv_1 : BOOL;
   Step_35_Conv_1 : BOOL;
   Step_36_Conv_1 : BOOL;
   Step_37_Conv_1 : BOOL;
   Step_38_Conv_1 : BOOL;
   Step_39_Conv_1 : BOOL;
   Step_40_Conv_1 : BOOL;
   Step_Alm_1 : DINT;
   Step_Conv_1 : DINT := 240;
   Storage1_YActualPosition : REAL := -649.99084;
   Storage1SeqToTec81 : DINT; {produced}
   Storage1toTec81 : DINT; {produced}
   Storage_PF_Conv_1 : BOOL;
   T_Conv_1_Sin_Pieza : TIMER;
   T_Conv_1_Step_00 : TIMER;
   T_Conv_1_Stop_Last_Time : TIMER;
   T_Fanuc_Pieza_Prensa_CNC : TIMER;
   T_FirstShot : TIMER;
   T_Permisive_Step_00 : TIMER;
   T_Permisive_Step_01 : TIMER;
   T_Permisive_Step_02 : TIMER;
   T_Permisive_Step_03 : TIMER;
   T_Permisive_Step_04 : TIMER;
   T_Permisive_Step_04_A : TIMER;
   T_Permisive_Step_05 : TIMER;
   T_Permisive_Step_06 : TIMER;
   T_Permisive_Step_07 : TIMER;
   T_Permisive_Step_08 : TIMER;
   T_Permisive_Step_09 : TIMER;
   T_Permisive_Step_10 : TIMER;
   T_Permisive_Step_11 : TIMER;
   T_Permisive_Step_12 : TIMER;
   T_Permisive_Step_13 : TIMER;
   T_Permisive_Step_14 : TIMER;
   T_Permisive_Step_15 : TIMER;
   T_Permisive_Step_16 : TIMER;
   T_Permisive_Step_17 : TIMER;
   T_Permisive_Step_18 : TIMER;
   T_Permisive_Step_19 : TIMER;
   T_Permisive_Step_20 : TIMER;
   T_Permisive_Step_21 : TIMER;
   T_Permisive_Step_22 : TIMER;
   T_Permisive_Step_23 : TIMER;
   T_Permisive_Step_24 : TIMER;
   T_Permisive_Step_25 : TIMER;
   T_Permisive_Step_26 : TIMER;
   T_Permisive_Step_27 : TIMER;
   T_Permisive_Step_28 : TIMER;
   T_Permisive_Step_29 : TIMER;
   T_Permisive_Step_30 : TIMER;
   T_Permisive_Step_31 : TIMER;
   T_Permisive_Step_32 : TIMER;
   T_Permisive_Step_33 : TIMER;
   T_Permisive_Step_34 : TIMER;
   T_Permisive_Step_35 : TIMER;
   T_Permisive_Step_36 : TIMER;
   T_Permisive_Step_37 : TIMER;
   T_Permisive_Step_38 : TIMER;
   T_Permisive_Step_39 : TIMER;
   T_Permisive_Step_40 : TIMER;
   T_Permissive_HomeStep1 : TIMER;
   T_Permissive_HomeStep2 : TIMER;
   T_Permissive_HomeStep3 : TIMER;
   T_Permissive_HomeStep4 : TIMER;
   T_Permissive_HomeStep5 : TIMER;
   T_Permissive_HomeStep6 : TIMER;
   T_Permissive_HomeStep7 : TIMER;
   T_Permissive_HomeStep8 : TIMER;
   T_Permissive_HomeStep9 : TIMER;
   T_Permissive_HomStep0 : TIMER;
   T_Pieza_Antes_Marcadora : TIMER;
   T_Pieza_Camara : TIMER;
   T_Pieza_FinDeCarrera : TIMER;
   T_Pieza_FinDeCarrera_Error : TIMER;
   T_Pieza_FinDeCarrera_Salida : TIMER;
   T_Pieza_Marcadora : TIMER;
   T_Pieza_MarcadoraTerminada : TIMER;
   T_Pieza_TomaFanuc : TIMER;
   Test_Bit : DINT := 537136129;
   Timer_1 : TIMER;
   Timer_2 : TIMER;
   Timer_3 : TIMER;
   Timer_4 : TIMER;
   Timer_5 : TIMER;
   Timer_6 : TIMER;
   Timer_7 : TIMER;
   Timer_8 : TIMER;
   To_Pos_Alm_1 : DINT; {produced}
   Tope_CNC_Conv_1 : BOOL;   // Tope Pistón CNC (Freno 5) Conveyor 1
   Tope_CNC_Conv_2 : BOOL;   // Tope Pistón CNC (Freno 5) Conveyor 2
   Tope_Marcadora_Conv_1 : BOOL;   // Tope Pistón Marcadora Láser (Freno 6) Conveyor 1
   Tope_Marcadora_Conv_2 : BOOL;   // Tope Pistón Marcadora Láser (Freno 6) Conveyor 2
   Tope_Salida_PH_Conv_1 : BOOL;   // Tope Pistón Salida de Producto (Freno 8) Conveyor 1
   Tope_Salida_PH_Conv_2 : BOOL;   // Tope Pistón Salida de Producto (Freno 8) Conveyor 2
   Tope_Vision_Conv_1 : BOOL;   // Tope Pistón Cáma de Visión Conveyor 1
   Tope_Vision_Conv_2 : BOOL;   // Tope Pistón Cámara de Visión Conveyor 2
   Usar_Proceso_CNC_1_de_Conveyor_1 : BOOL;   // Bit Para usar pasos del Robot Fanuc en el Conveyor 1
   X_Negative : BOOL;
   X_Positive : BOOL := 1;
   Y_Negative : BOOL := 1;
   Y_Positive : BOOL;
   Yaw_Negative : BOOL := 1;
   Yaw_Positive : BOOL;
   Yellow_Light_Alm_1 : BOOL := 1;
   Yellow_Light_Alm_2 : BOOL;
END_VAR

PROGRAM _02_Conveyor_1
VAR
   CamOnline : BOOL := 1;
   CompletedNS : BOOL;
   Count1 : COUNTER;
   Inspecting : BOOL;
   JobPass : BOOL;
   Timer : TIMER; {access Read Only}
   Timer1 : TIMER;
   Timer2 : TIMER;
   Timer3 : TIMER;
   Timer5 : TIMER; {access Read Only}
   trigger : BOOL := 1;
   TriggerGus1 : BOOL;
   TriggerGusEN : BOOL := 1;
   Valid : BOOL;
END_VAR
END_PROGRAM

PROGRAM MainProgram   (* main routine MainRoutine *)
VAR
   Contador : COUNTER;
   mem1 : BOOL;
   mem2 : BOOL := 1;
   mem3 : BOOL;
   mem4 : BOOL;
   mem5 : BOOL;
   PosDer_Alm_0_C : BOOL;
   PosDer_Alm_0_E : BOOL;
   PosDer_Alm_1_C : BOOL;
   PosDer_Alm_1_E : BOOL;
   PosDer_Alm_2_C : BOOL;
   PosDer_Alm_2_E : BOOL;
   PosDer_Alm_3_C : BOOL;
   PosDer_Alm_3_E : BOOL;
   PosDer_Alm_4_C : BOOL;
   PosDer_Alm_4_E : BOOL;
   PosDer_Alm_5_C : BOOL;
   PosDer_Alm_5_E : BOOL;
   PosIzq_Alm_0_C : BOOL;
   PosIzq_Alm_0_E : BOOL;
   PosIzq_Alm_1_C : BOOL;
   PosIzq_Alm_1_E : BOOL;
   PosIzq_Alm_2_C : BOOL;
   PosIzq_Alm_2_E : BOOL;
   PosIzq_Alm_3_C : BOOL;
   PosIzq_Alm_3_E : BOOL;
   PosIzq_Alm_4_C : BOOL;
   PosIzq_Alm_4_E : BOOL;
   PosIzq_Alm_5_C : BOOL;
   PosIzq_Alm_5_E : BOOL;
   TEMP1 : TIMER;
   TIM2 : TIMER;
   TIM3 : TIMER;
   TIM4 : TIMER;
END_VAR

ROUTINE Almacen1   (* ladder *)
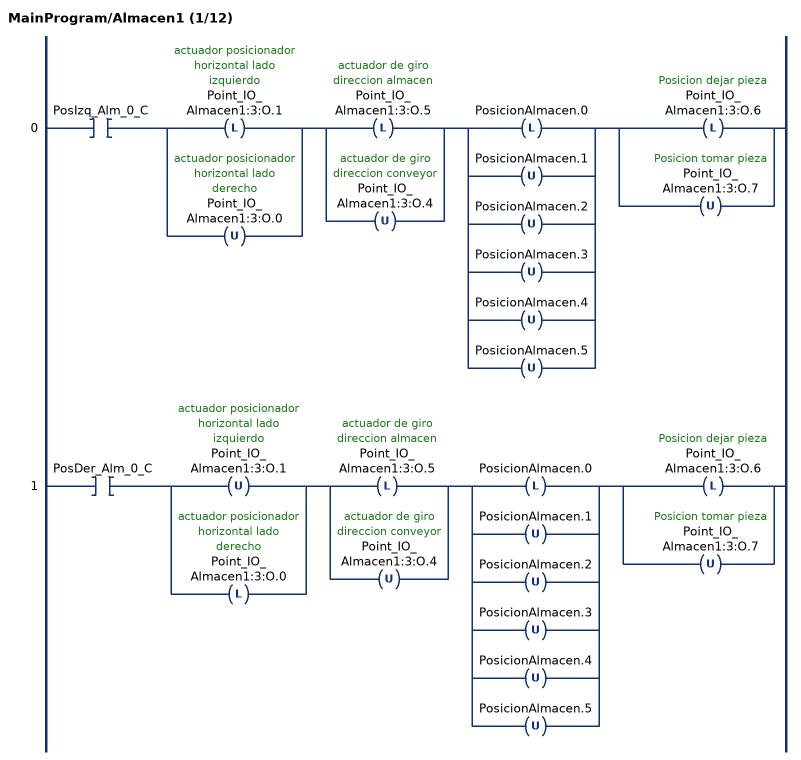
   0: XIC(PosIzq_Alm_0_C)[OTL(Point_IO_Almacen1:3:O.1) ,OTU(Point_IO_Almacen1:3:O.0) ][OTL(Point_IO_Almacen1:3:O.5) ,OTU(Point_IO_Almacen1:3:O.4) ][OTL(PosicionAlmacen.0) ,OTU(PosicionAlmacen.1) ,OTU(PosicionAlmacen.2) ,OTU(PosicionAlmacen.3) ,OTU(PosicionAlmacen.4) ,OTU(PosicionAlmacen.5) ][OTL(Point_IO_Almacen1:3:O.6) ,OTU(Point_IO_Almacen1:3:O.7) ];
   1: XIC(PosDer_Alm_0_C)[OTU(Point_IO_Almacen1:3:O.1) ,OTL(Point_IO_Almacen1:3:O.0) ][OTL(Point_IO_Almacen1:3:O.5) ,OTU(Point_IO_Almacen1:3:O.4) ][OTL(PosicionAlmacen.0) ,OTU(PosicionAlmacen.1) ,OTU(PosicionAlmacen.2) ,OTU(PosicionAlmacen.3) ,OTU(PosicionAlmacen.4) ,OTU(PosicionAlmacen.5) ][OTL(Point_IO_Almacen1:3:O.6) ,OTU(Point_IO_Almacen1:3:O.7) ];
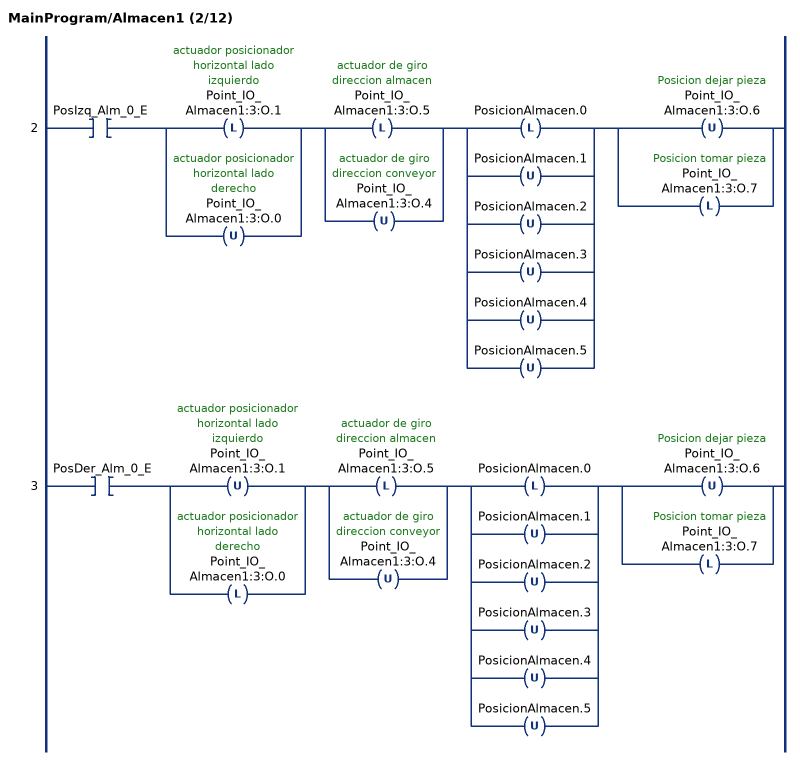
   2: XIC(PosIzq_Alm_0_E)[OTL(Point_IO_Almacen1:3:O.1) ,OTU(Point_IO_Almacen1:3:O.0) ][OTL(Point_IO_Almacen1:3:O.5) ,OTU(Point_IO_Almacen1:3:O.4) ][OTL(PosicionAlmacen.0) ,OTU(PosicionAlmacen.1) ,OTU(PosicionAlmacen.2) ,OTU(PosicionAlmacen.3) ,OTU(PosicionAlmacen.4) ,OTU(PosicionAlmacen.5) ][OTU(Point_IO_Almacen1:3:O.6) ,OTL(Point_IO_Almacen1:3:O.7) ];
   3: XIC(PosDer_Alm_0_E)[OTU(Point_IO_Almacen1:3:O.1) ,OTL(Point_IO_Almacen1:3:O.0) ][OTL(Point_IO_Almacen1:3:O.5) ,OTU(Point_IO_Almacen1:3:O.4) ][OTL(PosicionAlmacen.0) ,OTU(PosicionAlmacen.1) ,OTU(PosicionAlmacen.2) ,OTU(PosicionAlmacen.3) ,OTU(PosicionAlmacen.4) ,OTU(PosicionAlmacen.5) ][OTU(Point_IO_Almacen1:3:O.6) ,OTL(Point_IO_Almacen1:3:O.7) ];
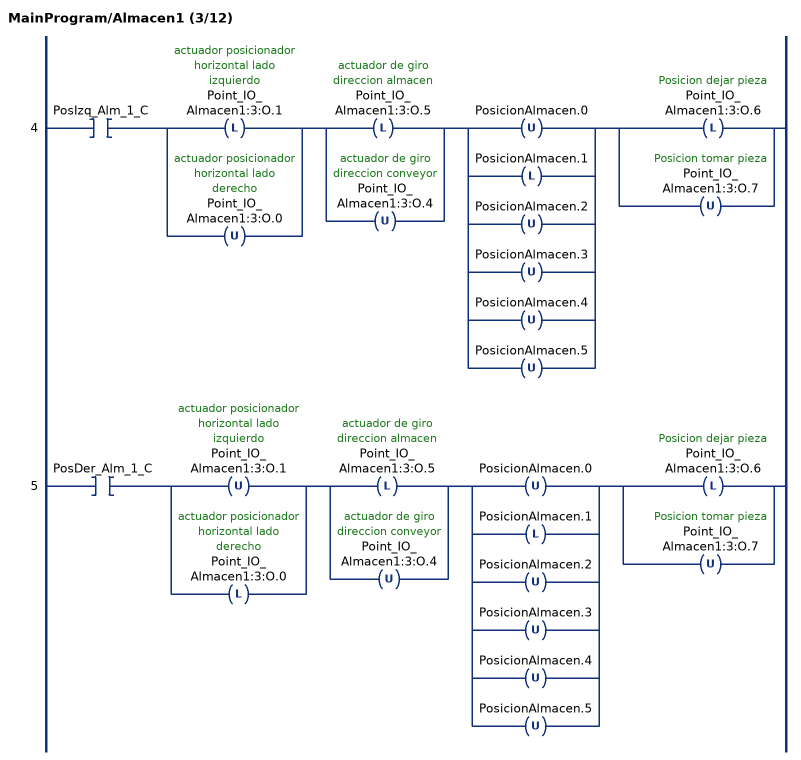
   4: XIC(PosIzq_Alm_1_C)[OTL(Point_IO_Almacen1:3:O.1) ,OTU(Point_IO_Almacen1:3:O.0) ][OTL(Point_IO_Almacen1:3:O.5) ,OTU(Point_IO_Almacen1:3:O.4) ][OTU(PosicionAlmacen.0) ,OTL(PosicionAlmacen.1) ,OTU(PosicionAlmacen.2) ,OTU(PosicionAlmacen.3) ,OTU(PosicionAlmacen.4) ,OTU(PosicionAlmacen.5) ][OTL(Point_IO_Almacen1:3:O.6) ,OTU(Point_IO_Almacen1:3:O.7) ];
   5: XIC(PosDer_Alm_1_C)[OTU(Point_IO_Almacen1:3:O.1) ,OTL(Point_IO_Almacen1:3:O.0) ][OTL(Point_IO_Almacen1:3:O.5) ,OTU(Point_IO_Almacen1:3:O.4) ][OTU(PosicionAlmacen.0) ,OTL(PosicionAlmacen.1) ,OTU(PosicionAlmacen.2) ,OTU(PosicionAlmacen.3) ,OTU(PosicionAlmacen.4) ,OTU(PosicionAlmacen.5) ][OTL(Point_IO_Almacen1:3:O.6) ,OTU(Point_IO_Almacen1:3:O.7) ];
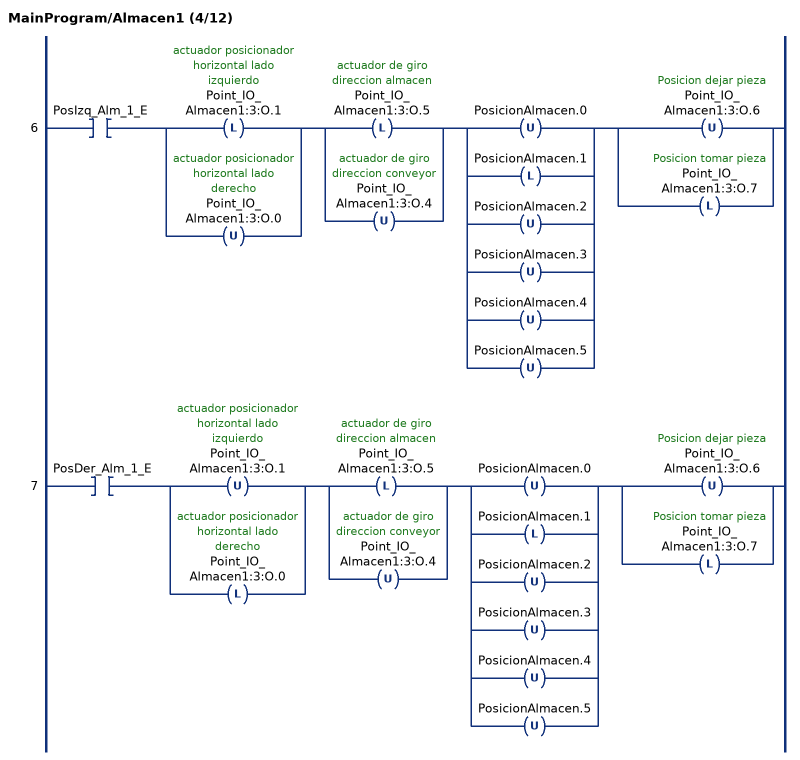
   6: XIC(PosIzq_Alm_1_E)[OTL(Point_IO_Almacen1:3:O.1) ,OTU(Point_IO_Almacen1:3:O.0) ][OTL(Point_IO_Almacen1:3:O.5) ,OTU(Point_IO_Almacen1:3:O.4) ][OTU(PosicionAlmacen.0) ,OTL(PosicionAlmacen.1) ,OTU(PosicionAlmacen.2) ,OTU(PosicionAlmacen.3) ,OTU(PosicionAlmacen.4) ,OTU(PosicionAlmacen.5) ][OTU(Point_IO_Almacen1:3:O.6) ,OTL(Point_IO_Almacen1:3:O.7) ];
   7: XIC(PosDer_Alm_1_E)[OTU(Point_IO_Almacen1:3:O.1) ,OTL(Point_IO_Almacen1:3:O.0) ][OTL(Point_IO_Almacen1:3:O.5) ,OTU(Point_IO_Almacen1:3:O.4) ][OTU(PosicionAlmacen.0) ,OTL(PosicionAlmacen.1) ,OTU(PosicionAlmacen.2) ,OTU(PosicionAlmacen.3) ,OTU(PosicionAlmacen.4) ,OTU(PosicionAlmacen.5) ][OTU(Point_IO_Almacen1:3:O.6) ,OTL(Point_IO_Almacen1:3:O.7) ];
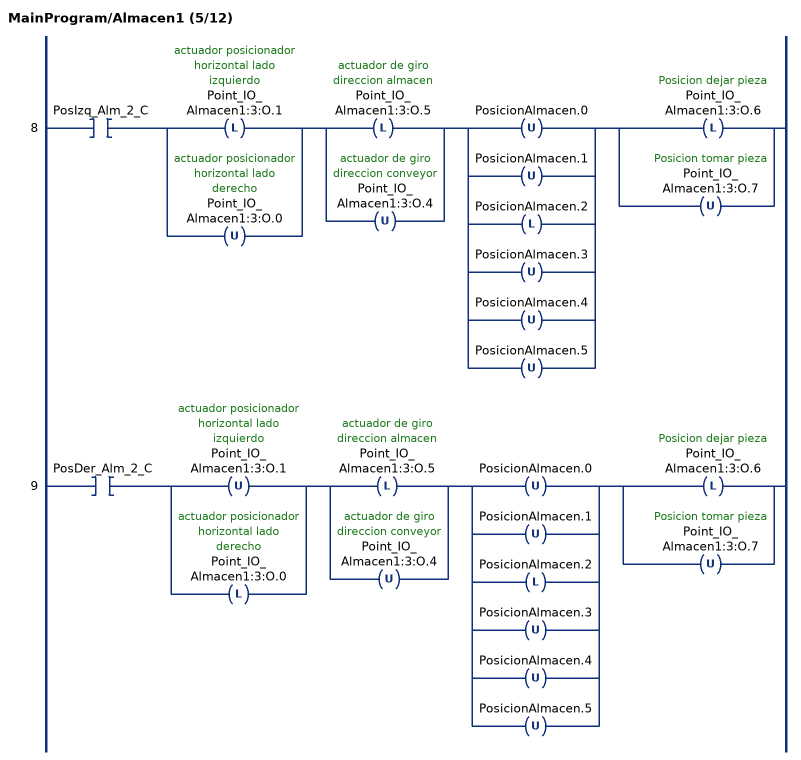
   8: XIC(PosIzq_Alm_2_C)[OTL(Point_IO_Almacen1:3:O.1) ,OTU(Point_IO_Almacen1:3:O.0) ][OTL(Point_IO_Almacen1:3:O.5) ,OTU(Point_IO_Almacen1:3:O.4) ][OTU(PosicionAlmacen.0) ,OTU(PosicionAlmacen.1) ,OTL(PosicionAlmacen.2) ,OTU(PosicionAlmacen.3) ,OTU(PosicionAlmacen.4) ,OTU(PosicionAlmacen.5) ][OTL(Point_IO_Almacen1:3:O.6) ,OTU(Point_IO_Almacen1:3:O.7) ];
   9: XIC(PosDer_Alm_2_C)[OTU(Point_IO_Almacen1:3:O.1) ,OTL(Point_IO_Almacen1:3:O.0) ][OTL(Point_IO_Almacen1:3:O.5) ,OTU(Point_IO_Almacen1:3:O.4) ][OTU(PosicionAlmacen.0) ,OTU(PosicionAlmacen.1) ,OTL(PosicionAlmacen.2) ,OTU(PosicionAlmacen.3) ,OTU(PosicionAlmacen.4) ,OTU(PosicionAlmacen.5) ][OTL(Point_IO_Almacen1:3:O.6) ,OTU(Point_IO_Almacen1:3:O.7) ];
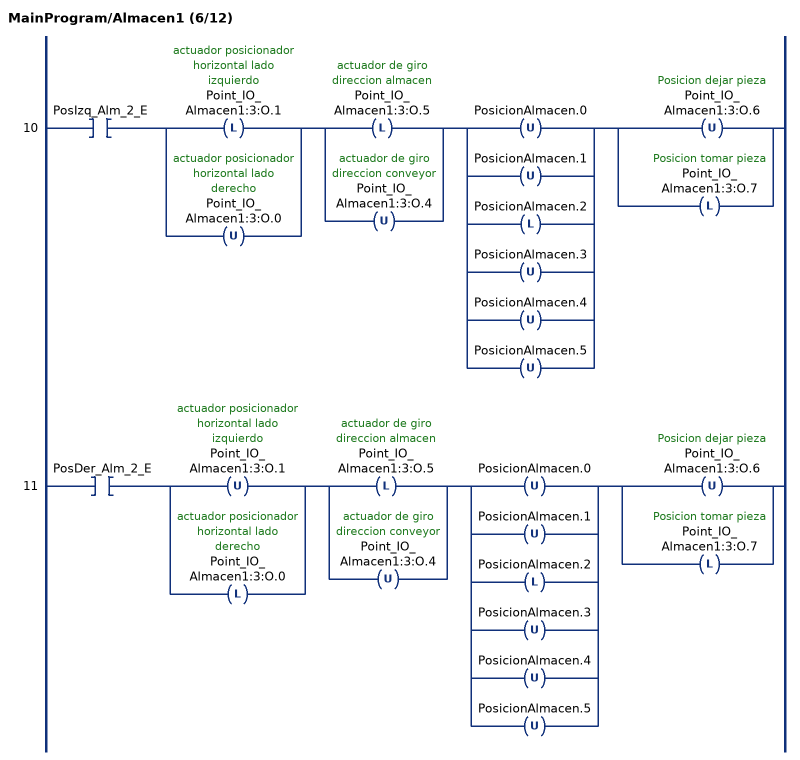
   10: XIC(PosIzq_Alm_2_E)[OTL(Point_IO_Almacen1:3:O.1) ,OTU(Point_IO_Almacen1:3:O.0) ][OTL(Point_IO_Almacen1:3:O.5) ,OTU(Point_IO_Almacen1:3:O.4) ][OTU(PosicionAlmacen.0) ,OTU(PosicionAlmacen.1) ,OTL(PosicionAlmacen.2) ,OTU(PosicionAlmacen.3) ,OTU(PosicionAlmacen.4) ,OTU(PosicionAlmacen.5) ][OTU(Point_IO_Almacen1:3:O.6) ,OTL(Point_IO_Almacen1:3:O.7) ];
   11: XIC(PosDer_Alm_2_E)[OTU(Point_IO_Almacen1:3:O.1) ,OTL(Point_IO_Almacen1:3:O.0) ][OTL(Point_IO_Almacen1:3:O.5) ,OTU(Point_IO_Almacen1:3:O.4) ][OTU(PosicionAlmacen.0) ,OTU(PosicionAlmacen.1) ,OTL(PosicionAlmacen.2) ,OTU(PosicionAlmacen.3) ,OTU(PosicionAlmacen.4) ,OTU(PosicionAlmacen.5) ][OTU(Point_IO_Almacen1:3:O.6) ,OTL(Point_IO_Almacen1:3:O.7) ];
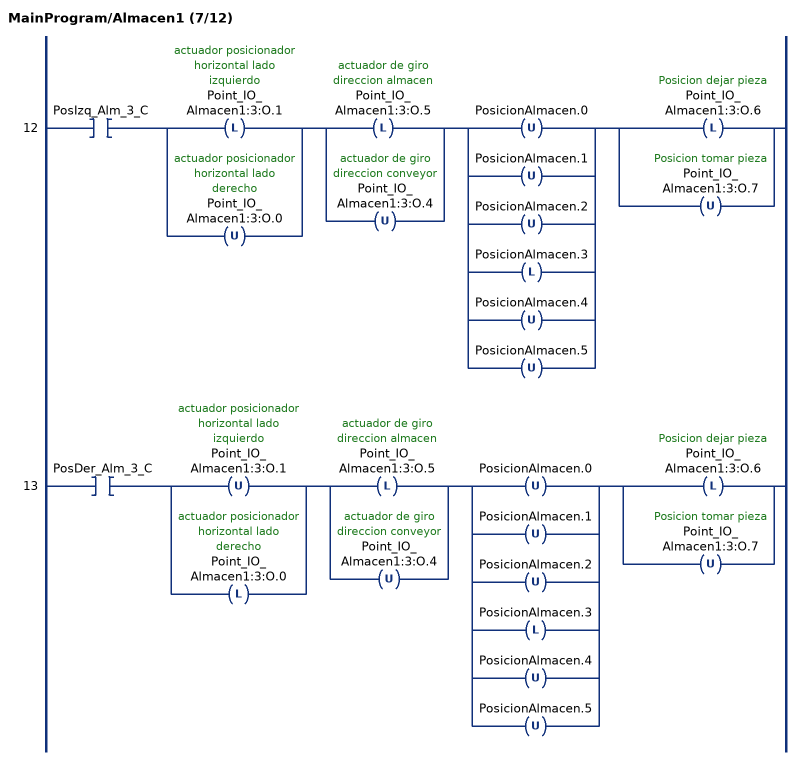
   12: XIC(PosIzq_Alm_3_C)[OTL(Point_IO_Almacen1:3:O.1) ,OTU(Point_IO_Almacen1:3:O.0) ][OTL(Point_IO_Almacen1:3:O.5) ,OTU(Point_IO_Almacen1:3:O.4) ][OTU(PosicionAlmacen.0) ,OTU(PosicionAlmacen.1) ,OTU(PosicionAlmacen.2) ,OTL(PosicionAlmacen.3) ,OTU(PosicionAlmacen.4) ,OTU(PosicionAlmacen.5) ][OTL(Point_IO_Almacen1:3:O.6) ,OTU(Point_IO_Almacen1:3:O.7) ];
   13: XIC(PosDer_Alm_3_C)[OTU(Point_IO_Almacen1:3:O.1) ,OTL(Point_IO_Almacen1:3:O.0) ][OTL(Point_IO_Almacen1:3:O.5) ,OTU(Point_IO_Almacen1:3:O.4) ][OTU(PosicionAlmacen.0) ,OTU(PosicionAlmacen.1) ,OTU(PosicionAlmacen.2) ,OTL(PosicionAlmacen.3) ,OTU(PosicionAlmacen.4) ,OTU(PosicionAlmacen.5) ][OTL(Point_IO_Almacen1:3:O.6) ,OTU(Point_IO_Almacen1:3:O.7) ];
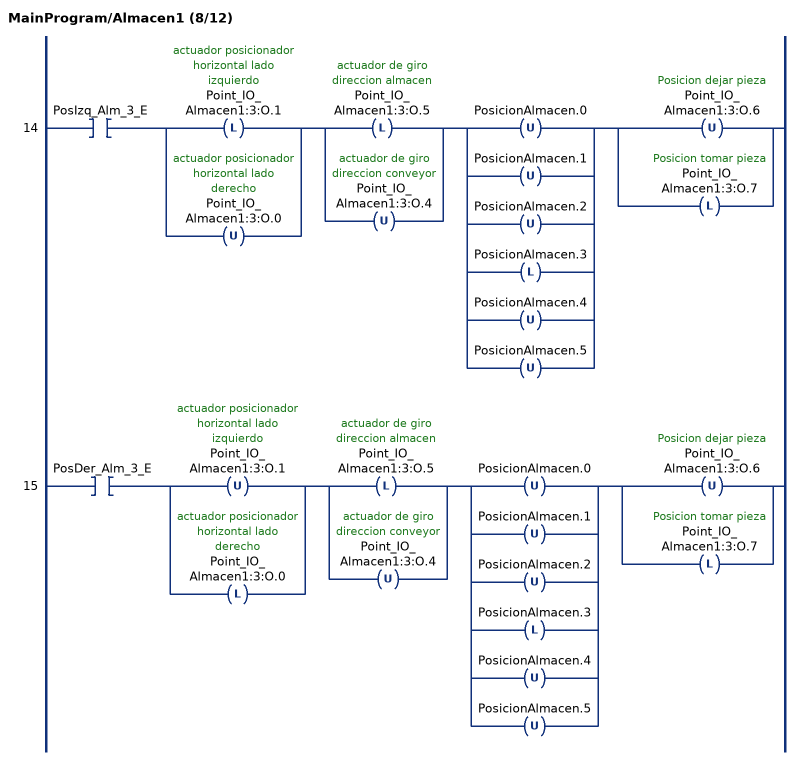
   14: XIC(PosIzq_Alm_3_E)[OTL(Point_IO_Almacen1:3:O.1) ,OTU(Point_IO_Almacen1:3:O.0) ][OTL(Point_IO_Almacen1:3:O.5) ,OTU(Point_IO_Almacen1:3:O.4) ][OTU(PosicionAlmacen.0) ,OTU(PosicionAlmacen.1) ,OTU(PosicionAlmacen.2) ,OTL(PosicionAlmacen.3) ,OTU(PosicionAlmacen.4) ,OTU(PosicionAlmacen.5) ][OTU(Point_IO_Almacen1:3:O.6) ,OTL(Point_IO_Almacen1:3:O.7) ];
   15: XIC(PosDer_Alm_3_E)[OTU(Point_IO_Almacen1:3:O.1) ,OTL(Point_IO_Almacen1:3:O.0) ][OTL(Point_IO_Almacen1:3:O.5) ,OTU(Point_IO_Almacen1:3:O.4) ][OTU(PosicionAlmacen.0) ,OTU(PosicionAlmacen.1) ,OTU(PosicionAlmacen.2) ,OTL(PosicionAlmacen.3) ,OTU(PosicionAlmacen.4) ,OTU(PosicionAlmacen.5) ][OTU(Point_IO_Almacen1:3:O.6) ,OTL(Point_IO_Almacen1:3:O.7) ];
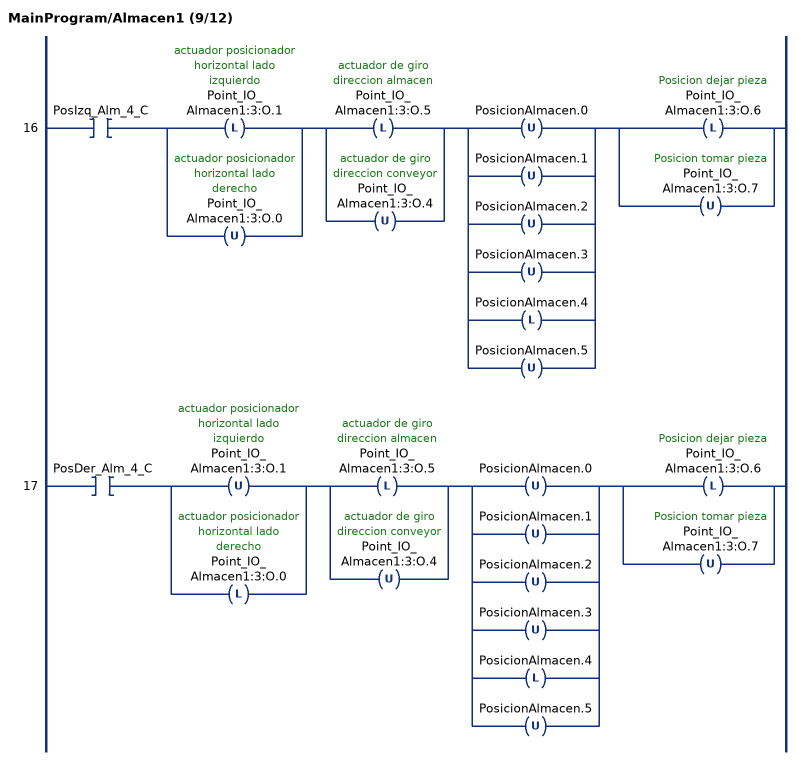
   16: XIC(PosIzq_Alm_4_C)[OTL(Point_IO_Almacen1:3:O.1) ,OTU(Point_IO_Almacen1:3:O.0) ][OTL(Point_IO_Almacen1:3:O.5) ,OTU(Point_IO_Almacen1:3:O.4) ][OTU(PosicionAlmacen.0) ,OTU(PosicionAlmacen.1) ,OTU(PosicionAlmacen.2) ,OTU(PosicionAlmacen.3) ,OTL(PosicionAlmacen.4) ,OTU(PosicionAlmacen.5) ][OTL(Point_IO_Almacen1:3:O.6) ,OTU(Point_IO_Almacen1:3:O.7) ];
   17: XIC(PosDer_Alm_4_C)[OTU(Point_IO_Almacen1:3:O.1) ,OTL(Point_IO_Almacen1:3:O.0) ][OTL(Point_IO_Almacen1:3:O.5) ,OTU(Point_IO_Almacen1:3:O.4) ][OTU(PosicionAlmacen.0) ,OTU(PosicionAlmacen.1) ,OTU(PosicionAlmacen.2) ,OTU(PosicionAlmacen.3) ,OTL(PosicionAlmacen.4) ,OTU(PosicionAlmacen.5) ][OTL(Point_IO_Almacen1:3:O.6) ,OTU(Point_IO_Almacen1:3:O.7) ];
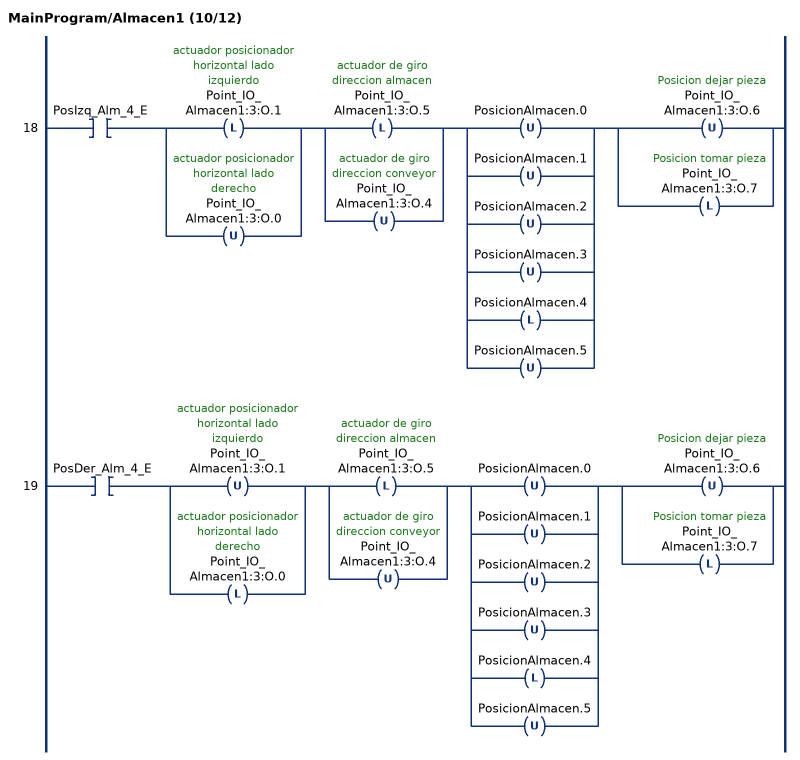
   18: XIC(PosIzq_Alm_4_E)[OTL(Point_IO_Almacen1:3:O.1) ,OTU(Point_IO_Almacen1:3:O.0) ][OTL(Point_IO_Almacen1:3:O.5) ,OTU(Point_IO_Almacen1:3:O.4) ][OTU(PosicionAlmacen.0) ,OTU(PosicionAlmacen.1) ,OTU(PosicionAlmacen.2) ,OTU(PosicionAlmacen.3) ,OTL(PosicionAlmacen.4) ,OTU(PosicionAlmacen.5) ][OTU(Point_IO_Almacen1:3:O.6) ,OTL(Point_IO_Almacen1:3:O.7) ];
   19: XIC(PosDer_Alm_4_E)[OTU(Point_IO_Almacen1:3:O.1) ,OTL(Point_IO_Almacen1:3:O.0) ][OTL(Point_IO_Almacen1:3:O.5) ,OTU(Point_IO_Almacen1:3:O.4) ][OTU(PosicionAlmacen.0) ,OTU(PosicionAlmacen.1) ,OTU(PosicionAlmacen.2) ,OTU(PosicionAlmacen.3) ,OTL(PosicionAlmacen.4) ,OTU(PosicionAlmacen.5) ][OTU(Point_IO_Almacen1:3:O.6) ,OTL(Point_IO_Almacen1:3:O.7) ];
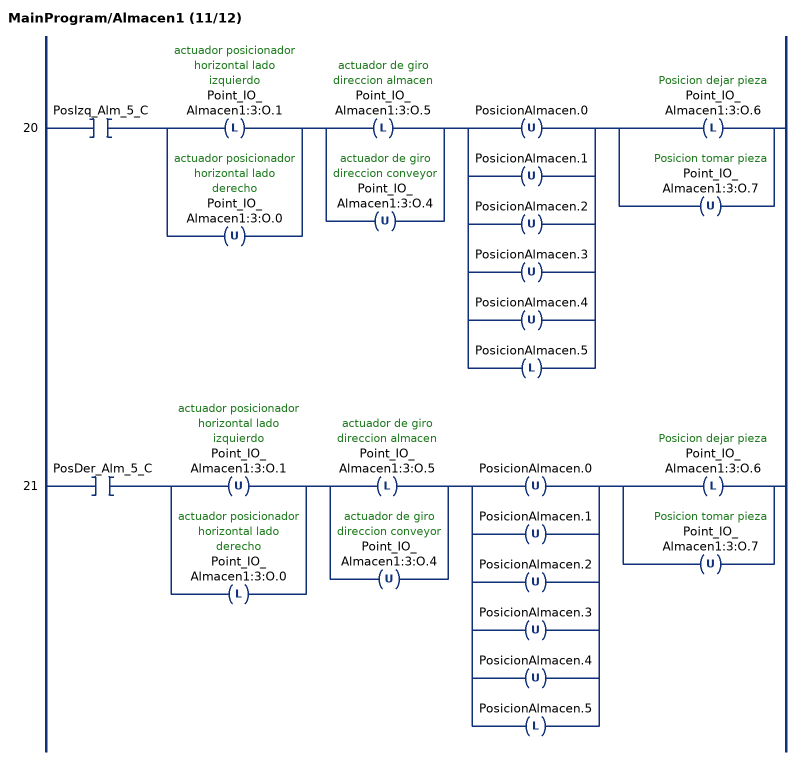
   20: XIC(PosIzq_Alm_5_C)[OTL(Point_IO_Almacen1:3:O.1) ,OTU(Point_IO_Almacen1:3:O.0) ][OTL(Point_IO_Almacen1:3:O.5) ,OTU(Point_IO_Almacen1:3:O.4) ][OTU(PosicionAlmacen.0) ,OTU(PosicionAlmacen.1) ,OTU(PosicionAlmacen.2) ,OTU(PosicionAlmacen.3) ,OTU(PosicionAlmacen.4) ,OTL(PosicionAlmacen.5) ][OTL(Point_IO_Almacen1:3:O.6) ,OTU(Point_IO_Almacen1:3:O.7) ];
   21: XIC(PosDer_Alm_5_C)[OTU(Point_IO_Almacen1:3:O.1) ,OTL(Point_IO_Almacen1:3:O.0) ][OTL(Point_IO_Almacen1:3:O.5) ,OTU(Point_IO_Almacen1:3:O.4) ][OTU(PosicionAlmacen.0) ,OTU(PosicionAlmacen.1) ,OTU(PosicionAlmacen.2) ,OTU(PosicionAlmacen.3) ,OTU(PosicionAlmacen.4) ,OTL(PosicionAlmacen.5) ][OTL(Point_IO_Almacen1:3:O.6) ,OTU(Point_IO_Almacen1:3:O.7) ];
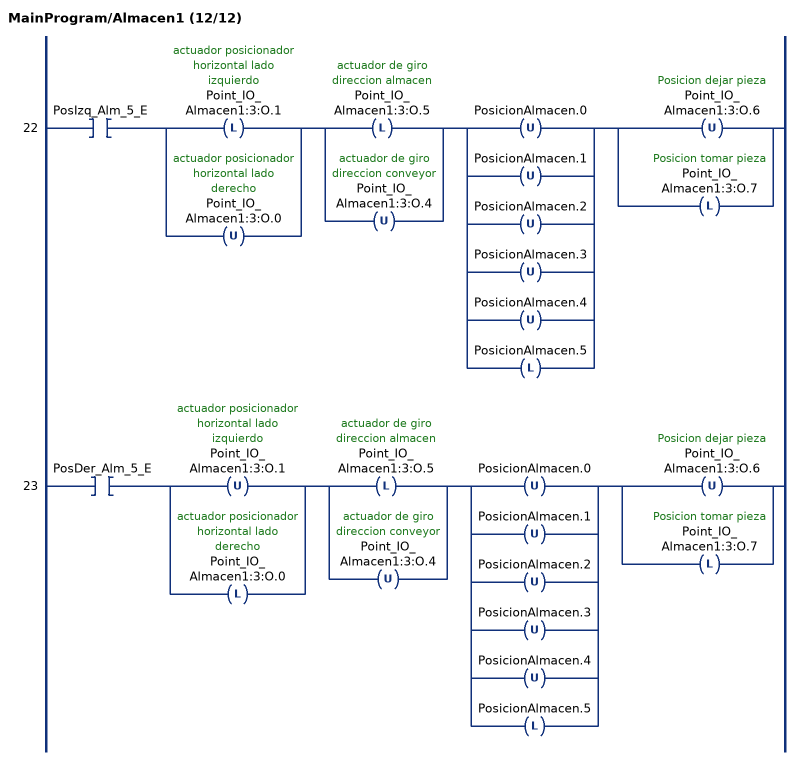
   22: XIC(PosIzq_Alm_5_E)[OTL(Point_IO_Almacen1:3:O.1) ,OTU(Point_IO_Almacen1:3:O.0) ][OTL(Point_IO_Almacen1:3:O.5) ,OTU(Point_IO_Almacen1:3:O.4) ][OTU(PosicionAlmacen.0) ,OTU(PosicionAlmacen.1) ,OTU(PosicionAlmacen.2) ,OTU(PosicionAlmacen.3) ,OTU(PosicionAlmacen.4) ,OTL(PosicionAlmacen.5) ][OTU(Point_IO_Almacen1:3:O.6) ,OTL(Point_IO_Almacen1:3:O.7) ];
   23: XIC(PosDer_Alm_5_E)[OTU(Point_IO_Almacen1:3:O.1) ,OTL(Point_IO_Almacen1:3:O.0) ][OTL(Point_IO_Almacen1:3:O.5) ,OTU(Point_IO_Almacen1:3:O.4) ][OTU(PosicionAlmacen.0) ,OTU(PosicionAlmacen.1) ,OTU(PosicionAlmacen.2) ,OTU(PosicionAlmacen.3) ,OTU(PosicionAlmacen.4) ,OTL(PosicionAlmacen.5) ][OTU(Point_IO_Almacen1:3:O.6) ,OTL(Point_IO_Almacen1:3:O.7) ];
END_ROUTINE

ROUTINE Camara_t   (* ladder *)
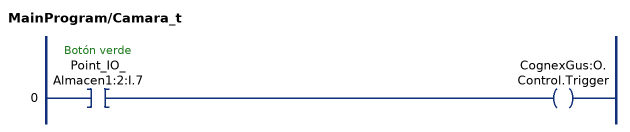
   0: XIC(Point_IO_Almacen1:2:I.7)OTE(CognexGus:O.Control.Trigger);
END_ROUTINE

ROUTINE MainRoutine   (* ladder *)
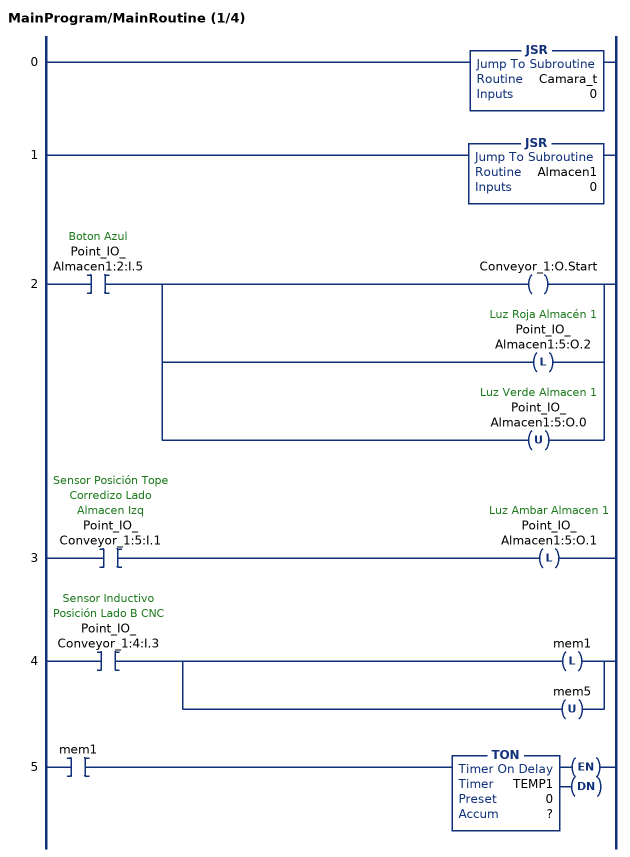
   0: JSR(Camara_t,0);
   1: JSR(Almacen1,0);
   2: XIC(Point_IO_Almacen1:2:I.5)[OTE(Conveyor_1:O.Start) ,OTL(Point_IO_Almacen1:5:O.2) ,OTU(Point_IO_Almacen1:5:O.0) ];
   3: XIC(Point_IO_Conveyor_1:5:I.1)OTL(Point_IO_Almacen1:5:O.1);
   4: XIC(Point_IO_Conveyor_1:4:I.3)[OTL(mem1) ,OTU(mem5) ];
   5: XIC(mem1)TON(TEMP1,?,?);
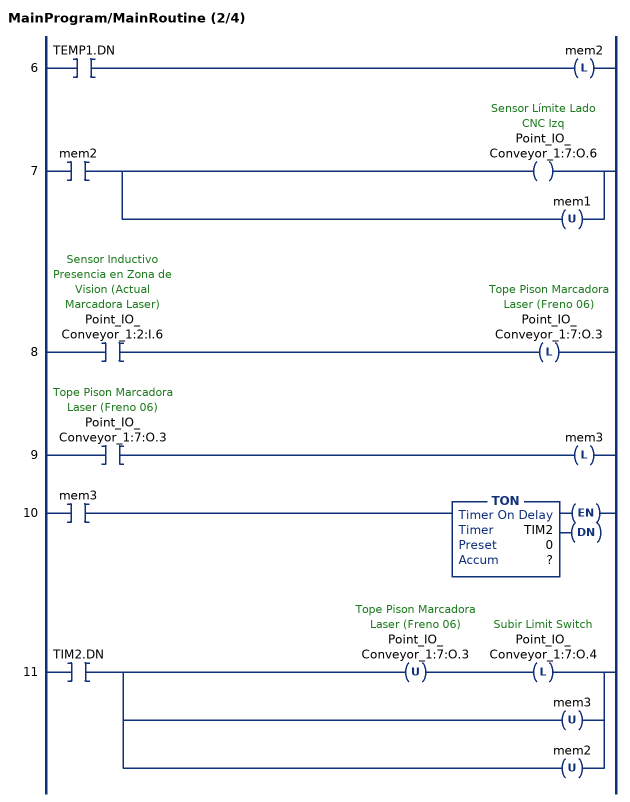
   6: XIC(TEMP1.DN)OTL(mem2);
   7: XIC(mem2)[OTE(Point_IO_Conveyor_1:7:O.6) ,OTU(mem1) ];
   8: XIC(Point_IO_Conveyor_1:2:I.6)OTL(Point_IO_Conveyor_1:7:O.3);
   9: XIC(Point_IO_Conveyor_1:7:O.3)OTL(mem3);
   10: XIC(mem3)TON(TIM2,?,?);
   11: XIC(TIM2.DN)[OTU(Point_IO_Conveyor_1:7:O.3) OTL(Point_IO_Conveyor_1:7:O.4) ,[OTU(mem3) ,OTU(mem2) ] ];
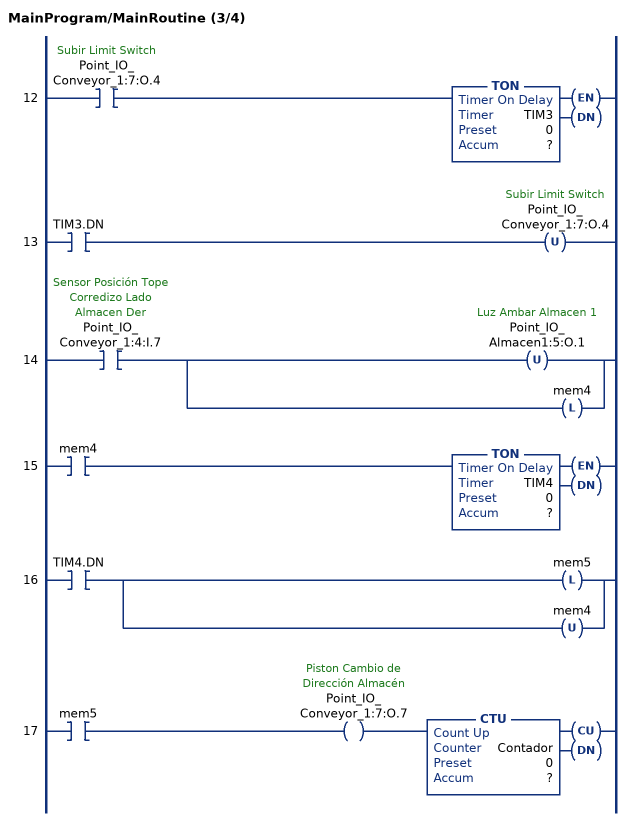
   12: XIC(Point_IO_Conveyor_1:7:O.4)TON(TIM3,?,?);
   13: XIC(TIM3.DN)OTU(Point_IO_Conveyor_1:7:O.4);
   14: XIC(Point_IO_Conveyor_1:4:I.7)[OTU(Point_IO_Almacen1:5:O.1) ,OTL(mem4) ];
   15: XIC(mem4)TON(TIM4,?,?);
   16: XIC(TIM4.DN)[OTL(mem5) ,OTU(mem4) ];
   17: XIC(mem5)OTE(Point_IO_Conveyor_1:7:O.7)CTU(Contador,?,?);
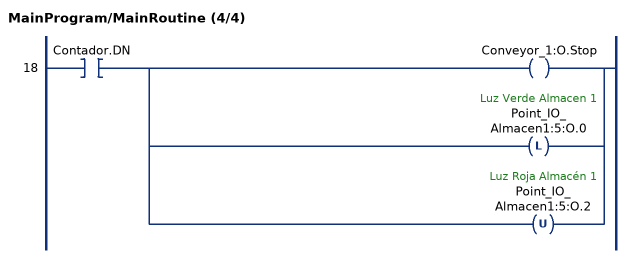
   18: XIC(Contador.DN)[OTE(Conveyor_1:O.Stop) ,OTL(Point_IO_Almacen1:5:O.0) ,OTU(Point_IO_Almacen1:5:O.2) ];
END_ROUTINE

ROUTINE Movimiento_elevador_alm1   (* ladder *)
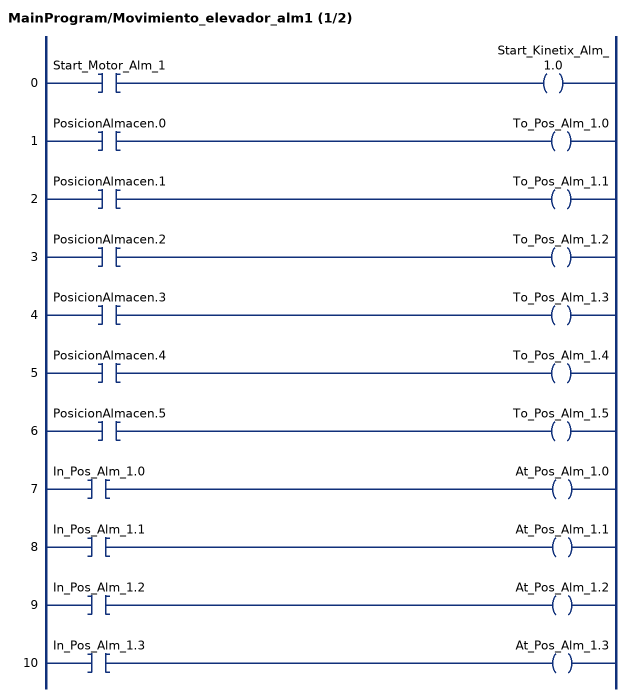
   0: XIC(Start_Motor_Alm_1)OTE(Start_Kinetix_Alm_1.0);
   1: XIC(PosicionAlmacen.0)OTE(To_Pos_Alm_1.0);
   2: XIC(PosicionAlmacen.1)OTE(To_Pos_Alm_1.1);
   3: XIC(PosicionAlmacen.2)OTE(To_Pos_Alm_1.2);
   4: XIC(PosicionAlmacen.3)OTE(To_Pos_Alm_1.3);
   5: XIC(PosicionAlmacen.4)OTE(To_Pos_Alm_1.4);
   6: XIC(PosicionAlmacen.5)OTE(To_Pos_Alm_1.5);
   7: XIC(In_Pos_Alm_1.0)OTE(At_Pos_Alm_1.0);
   8: XIC(In_Pos_Alm_1.1)OTE(At_Pos_Alm_1.1);
   9: XIC(In_Pos_Alm_1.2)OTE(At_Pos_Alm_1.2);
   10: XIC(In_Pos_Alm_1.3)OTE(At_Pos_Alm_1.3);
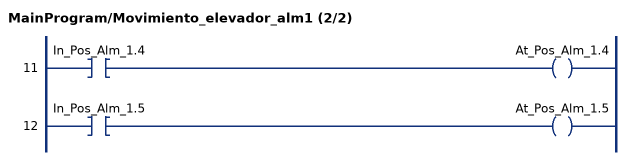
   11: XIC(In_Pos_Alm_1.4)OTE(At_Pos_Alm_1.4);
   12: XIC(In_Pos_Alm_1.5)OTE(At_Pos_Alm_1.5);
END_ROUTINE
END_PROGRAM

PROGRAM SafetyProgram   (* main routine MainRoutine, safety *)

ROUTINE MainRoutine   (* ladder *)
   0 (stored rung type 13): ;
END_ROUTINE
END_PROGRAM
